//     PlcTask Inputs/m01_rs3_r1._05_TT_01_Error <-> TC Channel 1/Status/Error
//     PlcTask Inputs/m01_rs3_r1._05_TT_03_Error <-> TC Channel 2/Status/Error
//     PlcTask Inputs/m01_rs3_r1._06_TT_01_Error <-> TC Channel 3/Status/Error
//     PlcTask Inputs/m01_rs3_r1._06_TT_03_Error <-> TC Channel 4/Status/Error
//     PlcTask Inputs/m01_rs3_r1._07_TT_01_Error <-> TC Channel 5/Status/Error
//     PlcTask Inputs/m01_rs3_r1._07_TT_03_Error <-> TC Channel 6/Status/Error
//     PlcTask Inputs/m01_rs3_r1._08_TT_01_Error <-> TC Channel 7/Status/Error
//     PlcTask Inputs/m01_rs3_r1._08_TT_03_Error <-> TC Channel 8/Status/Error
//   Phase0/Phase0 Instance <-> Device 4 (EtherCAT)/Term 1 Server Rack (EK1100)/Term 3 To DAC Mod and BOP PWR (EK1122)/Term 4 Main DAC Panel(EK1100)/Term 116 To RS3 (EK1122)/Term 117  RS3 INST Top Row (EK1100)/Term 144 (EL3318)
//     PlcTask Inputs/m01_rs3_r1._09_TT_01 <-> TC Channel 1/Value
//     PlcTask Inputs/m01_rs3_r1._09_TT_03 <-> TC Channel 2/Value
//     PlcTask Inputs/m01_rs3_r1._10_TT_01 <-> TC Channel 3/Value
//     PlcTask Inputs/m01_rs3_r1._10_TT_03 <-> TC Channel 4/Value
//     PlcTask Inputs/m01_rs3_r1._11_TT_01 <-> TC Channel 5/Value
//     PlcTask Inputs/m01_rs3_r1._11_TT_03 <-> TC Channel 6/Value
//     PlcTask Inputs/m01_rs3_r1._12_TT_01 <-> TC Channel 7/Value
//     PlcTask Inputs/m01_rs3_r1._12_TT_03 <-> TC Channel 8/Value
//     PlcTask Inputs/m01_rs3_r1._09_TT_01_Error <-> TC Channel 1/Status/Error
//     PlcTask Inputs/m01_rs3_r1._09_TT_03_Error <-> TC Channel 2/Status/Error
//     PlcTask Inputs/m01_rs3_r1._10_TT_01_Error <-> TC Channel 3/Status/Error
//     PlcTask Inputs/m01_rs3_r1._10_TT_03_Error <-> TC Channel 4/Status/Error
//     PlcTask Inputs/m01_rs3_r1._11_TT_01_Error <-> TC Channel 5/Status/Error
//     PlcTask Inputs/m01_rs3_r1._11_TT_03_Error <-> TC Channel 6/Status/Error
//     PlcTask Inputs/m01_rs3_r1._12_TT_01_Error <-> TC Channel 7/Status/Error
//     PlcTask Inputs/m01_rs3_r1._12_TT_03_Error <-> TC Channel 8/Status/Error
//   Phase0/Phase0 Instance <-> Device 4 (EtherCAT)/Term 1 Server Rack (EK1100)/Term 3 To DAC Mod and BOP PWR (EK1122)/Term 4 Main DAC Panel(EK1100)/Term 116 To RS3 (EK1122)/Term 117  RS3 INST Top Row (EK1100)/Term 145 (EL3318)
//     PlcTask Inputs/m01_rs3_r3._01_TT_01 <-> TC Channel 1/Value
//     PlcTask Inputs/m01_rs3_r3._01_TT_03 <-> TC Channel 2/Value
//     PlcTask Inputs/m01_rs3_r3._02_TT_01 <-> TC Channel 3/Value
//     PlcTask Inputs/m01_rs3_r3._02_TT_03 <-> TC Channel 4/Value
//     PlcTask Inputs/m01_rs3_r3._03_TT_01 <-> TC Channel 5/Value
//     PlcTask Inputs/m01_rs3_r3._03_TT_03 <-> TC Channel 6/Value
//     PlcTask Inputs/m01_rs3_r3._04_TT_01 <-> TC Channel 7/Value
//     PlcTask Inputs/m01_rs3_r3._04_TT_03 <-> TC Channel 8/Value
//     PlcTask Inputs/m01_rs3_r3._01_TT_01_Error <-> TC Channel 1/Status/Error
//     PlcTask Inputs/m01_rs3_r3._01_TT_03_Error <-> TC Channel 2/Status/Error
//     PlcTask Inputs/m01_rs3_r3._02_TT_01_Error <-> TC Channel 3/Status/Error
//     PlcTask Inputs/m01_rs3_r3._02_TT_03_Error <-> TC Channel 4/Status/Error
//     PlcTask Inputs/m01_rs3_r3._03_TT_01_Error <-> TC Channel 5/Status/Error
//     PlcTask Inputs/m01_rs3_r3._03_TT_03_Error <-> TC Channel 6/Status/Error
//     PlcTask Inputs/m01_rs3_r3._04_TT_01_Error <-> TC Channel 7/Status/Error
//     PlcTask Inputs/m01_rs3_r3._04_TT_03_Error <-> TC Channel 8/Status/Error
//   Phase0/Phase0 Instance <-> Device 4 (EtherCAT)/Term 1 Server Rack (EK1100)/Term 3 To DAC Mod and BOP PWR (EK1122)/Term 4 Main DAC Panel(EK1100)/Term 116 To RS3 (EK1122)/Term 117  RS3 INST Top Row (EK1100)/Term 146 (EL3318)
//     PlcTask Inputs/m01_rs3_r3._05_TT_01 <-> TC Channel 1/Value
//     PlcTask Inputs/m01_rs3_r3._05_TT_03 <-> TC Channel 2/Value
//     PlcTask Inputs/m01_rs3_r3._06_TT_01 <-> TC Channel 3/Value
//     PlcTask Inputs/m01_rs3_r3._06_TT_03 <-> TC Channel 4/Value
//     PlcTask Inputs/m01_rs3_r3._07_TT_01 <-> TC Channel 5/Value
//     PlcTask Inputs/m01_rs3_r3._07_TT_03 <-> TC Channel 6/Value
//     PlcTask Inputs/m01_rs3_r3._08_TT_01 <-> TC Channel 7/Value
//     PlcTask Inputs/m01_rs3_r3._08_TT_03 <-> TC Channel 8/Value
//     PlcTask Inputs/m01_rs3_r3._05_TT_01_Error <-> TC Channel 1/Status/Error
//     PlcTask Inputs/m01_rs3_r3._05_TT_03_Error <-> TC Channel 2/Status/Error
//     PlcTask Inputs/m01_rs3_r3._06_TT_01_Error <-> TC Channel 3/Status/Error
//     PlcTask Inputs/m01_rs3_r3._06_TT_03_Error <-> TC Channel 4/Status/Error
//     PlcTask Inputs/m01_rs3_r3._07_TT_01_Error <-> TC Channel 5/Status/Error
//     PlcTask Inputs/m01_rs3_r3._07_TT_03_Error <-> TC Channel 6/Status/Error
//     PlcTask Inputs/m01_rs3_r3._08_TT_01_Error <-> TC Channel 7/Status/Error
//     PlcTask Inputs/m01_rs3_r3._08_TT_03_Error <-> TC Channel 8/Status/Error
//   Phase0/Phase0 Instance <-> Device 4 (EtherCAT)/Term 1 Server Rack (EK1100)/Term 3 To DAC Mod and BOP PWR (EK1122)/Term 4 Main DAC Panel(EK1100)/Term 116 To RS3 (EK1122)/Term 117  RS3 INST Top Row (EK1100)/Term 147 (EL3318)
//     PlcTask Inputs/m01_rs3_r3._09_TT_01 <-> TC Channel 1/Value
//     PlcTask Inputs/m01_rs3_r3._09_TT_03 <-> TC Channel 2/Value
//     PlcTask Inputs/m01_rs3_r3._10_TT_01 <-> TC Channel 3/Value
//     PlcTask Inputs/m01_rs3_r3._10_TT_03 <-> TC Channel 4/Value
//     PlcTask Inputs/m01_rs3_r3._11_TT_01 <-> TC Channel 5/Value
//     PlcTask Inputs/m01_rs3_r3._11_TT_03 <-> TC Channel 6/Value
//     PlcTask Inputs/m01_rs3_r3._12_TT_01 <-> TC Channel 7/Value
//     PlcTask Inputs/m01_rs3_r3._12_TT_03 <-> TC Channel 8/Value
//     PlcTask Inputs/m01_rs3_r3._09_TT_01_Error <-> TC Channel 1/Status/Error
//     PlcTask Inputs/m01_rs3_r3._09_TT_03_Error <-> TC Channel 2/Status/Error
//     PlcTask Inputs/m01_rs3_r3._10_TT_01_Error <-> TC Channel 3/Status/Error
//     PlcTask Inputs/m01_rs3_r3._10_TT_03_Error <-> TC Channel 4/Status/Error
//     PlcTask Inputs/m01_rs3_r3._11_TT_01_Error <-> TC Channel 5/Status/Error
//     PlcTask Inputs/m01_rs3_r3._11_TT_03_Error <-> TC Channel 6/Status/Error
//     PlcTask Inputs/m01_rs3_r3._12_TT_01_Error <-> TC Channel 7/Status/Error
//     PlcTask Inputs/m01_rs3_r3._12_TT_03_Error <-> TC Channel 8/Status/Error
//   Phase0/Phase0 Instance <-> Device 4 (EtherCAT)/Term 1 Server Rack (EK1100)/Term 3 To DAC Mod and BOP PWR (EK1122)/Term 4 Main DAC Panel(EK1100)/Term 116 To RS3 (EK1122)/Term 117  RS3 INST Top Row (EK1100)/Term 149 (EL3318)
//     PlcTask Inputs/m01_rs3_r2._01_TT_01 <-> TC Channel 1/Value
//     PlcTask Inputs/m01_rs3_r2._01_TT_03 <-> TC Channel 2/Value
//     PlcTask Inputs/m01_rs3_r2._02_TT_01 <-> TC Channel 3/Value
//     PlcTask Inputs/m01_rs3_r2._02_TT_03 <-> TC Channel 4/Value
//     PlcTask Inputs/m01_rs3_r2._03_TT_01 <-> TC Channel 5/Value
//     PlcTask Inputs/m01_rs3_r2._03_TT_03 <-> TC Channel 6/Value
//     PlcTask Inputs/m01_rs3_r2._04_TT_01 <-> TC Channel 7/Value
//     PlcTask Inputs/m01_rs3_r2._04_TT_03 <-> TC Channel 8/Value
//     PlcTask Inputs/m01_rs3_r2._01_TT_01_Error <-> TC Channel 1/Status/Error
//     PlcTask Inputs/m01_rs3_r2._01_TT_03_Error <-> TC Channel 2/Status/Error
//     PlcTask Inputs/m01_rs3_r2._02_TT_01_Error <-> TC Channel 3/Status/Error
//     PlcTask Inputs/m01_rs3_r2._02_TT_03_Error <-> TC Channel 4/Status/Error
//     PlcTask Inputs/m01_rs3_r2._03_TT_01_Error <-> TC Channel 5/Status/Error
//     PlcTask Inputs/m01_rs3_r2._03_TT_03_Error <-> TC Channel 6/Status/Error
//     PlcTask Inputs/m01_rs3_r2._04_TT_01_Error <-> TC Channel 7/Status/Error
//     PlcTask Inputs/m01_rs3_r2._04_TT_03_Error <-> TC Channel 8/Status/Error
//   Phase0/Phase0 Instance <-> Device 4 (EtherCAT)/Term 1 Server Rack (EK1100)/Term 3 To DAC Mod and BOP PWR (EK1122)/Term 4 Main DAC Panel(EK1100)/Term 116 To RS3 (EK1122)/Term 117  RS3 INST Top Row (EK1100)/Term 150 (EL3318)
//     PlcTask Inputs/m01_rs3_r2._05_TT_01 <-> TC Channel 1/Value
//     PlcTask Inputs/m01_rs3_r2._05_TT_03 <-> TC Channel 2/Value
//     PlcTask Inputs/m01_rs3_r2._06_TT_01 <-> TC Channel 3/Value
//     PlcTask Inputs/m01_rs3_r2._06_TT_03 <-> TC Channel 4/Value
//     PlcTask Inputs/m01_rs3_r2._07_TT_01 <-> TC Channel 5/Value
//     PlcTask Inputs/m01_rs3_r2._07_TT_03 <-> TC Channel 6/Value
//     PlcTask Inputs/m01_rs3_r2._08_TT_01 <-> TC Channel 7/Value
//     PlcTask Inputs/m01_rs3_r2._08_TT_03 <-> TC Channel 8/Value
//     PlcTask Inputs/m01_rs3_r2._05_TT_01_Error <-> TC Channel 1/Status/Error
//     PlcTask Inputs/m01_rs3_r2._05_TT_03_Error <-> TC Channel 2/Status/Error
//     PlcTask Inputs/m01_rs3_r2._06_TT_01_Error <-> TC Channel 3/Status/Error
//     PlcTask Inputs/m01_rs3_r2._06_TT_03_Error <-> TC Channel 4/Status/Error
//     PlcTask Inputs/m01_rs3_r2._07_TT_01_Error <-> TC Channel 5/Status/Error
//     PlcTask Inputs/m01_rs3_r2._07_TT_03_Error <-> TC Channel 6/Status/Error
//     PlcTask Inputs/m01_rs3_r2._08_TT_01_Error <-> TC Channel 7/Status/Error
//     PlcTask Inputs/m01_rs3_r2._08_TT_03_Error <-> TC Channel 8/Status/Error
//   Phase0/Phase0 Instance <-> Device 4 (EtherCAT)/Term 1 Server Rack (EK1100)/Term 3 To DAC Mod and BOP PWR (EK1122)/Term 4 Main DAC Panel(EK1100)/Term 116 To RS3 (EK1122)/Term 117  RS3 INST Top Row (EK1100)/Term 151 (EL3318)
//     PlcTask Inputs/m01_rs3_r2._09_TT_01 <-> TC Channel 1/Value
//     PlcTask Inputs/m01_rs3_r2._09_TT_03 <-> TC Channel 2/Value
//     PlcTask Inputs/m01_rs3_r2._10_TT_01 <-> TC Channel 3/Value
//     PlcTask Inputs/m01_rs3_r2._10_TT_03 <-> TC Channel 4/Value
//     PlcTask Inputs/m01_rs3_r2._11_TT_01 <-> TC Channel 5/Value
//     PlcTask Inputs/m01_rs3_r2._11_TT_03 <-> TC Channel 6/Value
//     PlcTask Inputs/m01_rs3_r2._12_TT_01 <-> TC Channel 7/Value
//     PlcTask Inputs/m01_rs3_r2._12_TT_03 <-> TC Channel 8/Value
//     PlcTask Inputs/m01_rs3_r2._09_TT_01_Error <-> TC Channel 1/Status/Error
//     PlcTask Inputs/m01_rs3_r2._09_TT_03_Error <-> TC Channel 2/Status/Error
//     PlcTask Inputs/m01_rs3_r2._10_TT_01_Error <-> TC Channel 3/Status/Error
//     PlcTask Inputs/m01_rs3_r2._10_TT_03_Error <-> TC Channel 4/Status/Error
//     PlcTask Inputs/m01_rs3_r2._11_TT_01_Error <-> TC Channel 5/Status/Error
//     PlcTask Inputs/m01_rs3_r2._11_TT_03_Error <-> TC Channel 6/Status/Error
//     PlcTask Inputs/m01_rs3_r2._12_TT_01_Error <-> TC Channel 7/Status/Error
//     PlcTask Inputs/m01_rs3_r2._12_TT_03_Error <-> TC Channel 8/Status/Error
//   Phase0/Phase0 Instance <-> Device 4 (EtherCAT)/Term 1 Server Rack (EK1100)/Term 3 To DAC Mod and BOP PWR (EK1122)/Term 4 Main DAC Panel(EK1100)/Term 116 To RS3 (EK1122)/Term 117  RS3 INST Top Row (EK1100)/Term 152 (EL3318)
//     PlcTask Inputs/m01_rs3_r4._01_TT_01 <-> TC Channel 1/Value
//     PlcTask Inputs/m01_rs3_r4._01_TT_03 <-> TC Channel 2/Value
//     PlcTask Inputs/m01_rs3_r4._02_TT_01 <-> TC Channel 3/Value
//     PlcTask Inputs/m01_rs3_r4._02_TT_03 <-> TC Channel 4/Value
//     PlcTask Inputs/m01_rs3_r4._03_TT_01 <-> TC Channel 5/Value
//     PlcTask Inputs/m01_rs3_r4._03_TT_03 <-> TC Channel 6/Value
//     PlcTask Inputs/m01_rs3_r4._04_TT_01 <-> TC Channel 7/Value
//     PlcTask Inputs/m01_rs3_r4._04_TT_03 <-> TC Channel 8/Value
//     PlcTask Inputs/m01_rs3_r4._01_TT_01_Error <-> TC Channel 1/Status/Error
//     PlcTask Inputs/m01_rs3_r4._01_TT_03_Error <-> TC Channel 2/Status/Error
//     PlcTask Inputs/m01_rs3_r4._02_TT_01_Error <-> TC Channel 3/Status/Error
//     PlcTask Inputs/m01_rs3_r4._02_TT_03_Error <-> TC Channel 4/Status/Error
//     PlcTask Inputs/m01_rs3_r4._03_TT_01_Error <-> TC Channel 5/Status/Error
//     PlcTask Inputs/m01_rs3_r4._03_TT_03_Error <-> TC Channel 6/Status/Error
//     PlcTask Inputs/m01_rs3_r4._04_TT_01_Error <-> TC Channel 7/Status/Error
//     PlcTask Inputs/m01_rs3_r4._04_TT_03_Error <-> TC Channel 8/Status/Error
//   Phase0/Phase0 Instance <-> Device 4 (EtherCAT)/Term 1 Server Rack (EK1100)/Term 3 To DAC Mod and BOP PWR (EK1122)/Term 4 Main DAC Panel(EK1100)/Term 116 To RS3 (EK1122)/Term 117  RS3 INST Top Row (EK1100)/Term 153 (EL3318)
//     PlcTask Inputs/m01_rs3_r4._05_TT_01 <-> TC Channel 1/Value
//     PlcTask Inputs/m01_rs3_r4._05_TT_03 <-> TC Channel 2/Value
//     PlcTask Inputs/m01_rs3_r4._06_TT_01 <-> TC Channel 3/Value
//     PlcTask Inputs/m01_rs3_r4._06_TT_03 <-> TC Channel 4/Value
//     PlcTask Inputs/m01_rs3_r4._07_TT_01 <-> TC Channel 5/Value
//     PlcTask Inputs/m01_rs3_r4._07_TT_03 <-> TC Channel 6/Value
//     PlcTask Inputs/m01_rs3_r4._08_TT_01 <-> TC Channel 7/Value
//     PlcTask Inputs/m01_rs3_r4._08_TT_03 <-> TC Channel 8/Value
//     PlcTask Inputs/m01_rs3_r4._05_TT_01_Error <-> TC Channel 1/Status/Error
//     PlcTask Inputs/m01_rs3_r4._05_TT_03_Error <-> TC Channel 2/Status/Error
//     PlcTask Inputs/m01_rs3_r4._06_TT_01_Error <-> TC Channel 3/Status/Error
//     PlcTask Inputs/m01_rs3_r4._06_TT_03_Error <-> TC Channel 4/Status/Error
//     PlcTask Inputs/m01_rs3_r4._07_TT_01_Error <-> TC Channel 5/Status/Error
//     PlcTask Inputs/m01_rs3_r4._07_TT_03_Error <-> TC Channel 6/Status/Error
//     PlcTask Inputs/m01_rs3_r4._08_TT_01_Error <-> TC Channel 7/Status/Error
//     PlcTask Inputs/m01_rs3_r4._08_TT_03_Error <-> TC Channel 8/Status/Error
//   Phase0/Phase0 Instance <-> Device 4 (EtherCAT)/Term 1 Server Rack (EK1100)/Term 3 To DAC Mod and BOP PWR (EK1122)/Term 4 Main DAC Panel(EK1100)/Term 116 To RS3 (EK1122)/Term 117  RS3 INST Top Row (EK1100)/Term 154 (EL3318)
//     PlcTask Inputs/m01_rs3_r4._09_TT_01 <-> TC Channel 1/Value
//     PlcTask Inputs/m01_rs3_r4._09_TT_03 <-> TC Channel 2/Value
//     PlcTask Inputs/m01_rs3_r4._10_TT_01 <-> TC Channel 3/Value
//     PlcTask Inputs/m01_rs3_r4._10_TT_03 <-> TC Channel 4/Value
//     PlcTask Inputs/m01_rs3_r4._11_TT_01 <-> TC Channel 5/Value
//     PlcTask Inputs/m01_rs3_r4._11_TT_03 <-> TC Channel 6/Value
//     PlcTask Inputs/m01_rs3_r4._12_TT_01 <-> TC Channel 7/Value
//     PlcTask Inputs/m01_rs3_r4._12_TT_03 <-> TC Channel 8/Value
//     PlcTask Inputs/m01_rs3_r4._09_TT_01_Error <-> TC Channel 1/Status/Error
//     PlcTask Inputs/m01_rs3_r4._09_TT_03_Error <-> TC Channel 2/Status/Error
//     PlcTask Inputs/m01_rs3_r4._10_TT_01_Error <-> TC Channel 3/Status/Error
//     PlcTask Inputs/m01_rs3_r4._10_TT_03_Error <-> TC Channel 4/Status/Error
//     PlcTask Inputs/m01_rs3_r4._11_TT_01_Error <-> TC Channel 5/Status/Error
//     PlcTask Inputs/m01_rs3_r4._11_TT_03_Error <-> TC Channel 6/Status/Error
//     PlcTask Inputs/m01_rs3_r4._12_TT_01_Error <-> TC Channel 7/Status/Error
//     PlcTask Inputs/m01_rs3_r4._12_TT_03_Error <-> TC Channel 8/Status/Error
//   Phase0/Phase0 Instance <-> Device 4 (EtherCAT)/Term 1 Server Rack (EK1100)/Term 3 To DAC Mod and BOP PWR (EK1122)/Term 4 Main DAC Panel(EK1100)/Term 116 To RS3 (EK1122)/Term 117  RS3 INST Top Row (EK1100)/Term 156 (EL3214)
//     PlcTask Inputs/m01_rs3_r1.TT_05 <-> RTD Inputs Channel 1/Value
//     PlcTask Inputs/m01_rs3_r2.TT_05 <-> RTD Inputs Channel 3/Value
//     PlcTask Inputs/m01_rs3_r3.TT_05 <-> RTD Inputs Channel 2/Value
//     PlcTask Inputs/m01_rs3_r4.TT_05 <-> RTD Inputs Channel 4/Value
//     PlcTask Inputs/m01_rs3_r1.reactor_wall_temp_error <-> RTD Inputs Channel 1/Status/Error
//     PlcTask Inputs/m01_rs3_r2.reactor_wall_temp_error <-> RTD Inputs Channel 3/Status/Error
//     PlcTask Inputs/m01_rs3_r3.reactor_wall_temp_error <-> RTD Inputs Channel 2/Status/Error
//     PlcTask Inputs/m01_rs3_r4.reactor_wall_temp_error <-> RTD Inputs Channel 4/Status/Error
//   Phase0/Phase0 Instance <-> Device 4 (EtherCAT)/Term 1 Server Rack (EK1100)/Term 3 To DAC Mod and BOP PWR (EK1122)/Term 4 Main DAC Panel(EK1100)/Term 116 To RS3 (EK1122)/Term 117  RS3 INST Top Row (EK1100)/Term 157 (EL3214)
//     PlcTask Inputs/m01_rs3_r1.TT_06 <-> RTD Inputs Channel 1/Value
//     PlcTask Inputs/m01_rs3_r2.TT_06 <-> RTD Inputs Channel 3/Value
//     PlcTask Inputs/m01_rs3_r3.TT_06 <-> RTD Inputs Channel 2/Value
//     PlcTask Inputs/m01_rs3_r4.TT_06 <-> RTD Inputs Channel 4/Value
//     PlcTask Inputs/m01_rs3_r1.outlet_line_temp_error <-> RTD Inputs Channel 1/Status/Error
//     PlcTask Inputs/m01_rs3_r2.outlet_line_temp_error <-> RTD Inputs Channel 3/Status/Error
//     PlcTask Inputs/m01_rs3_r3.outlet_line_temp_error <-> RTD Inputs Channel 2/Status/Error
//     PlcTask Inputs/m01_rs3_r4.outlet_line_temp_error <-> RTD Inputs Channel 4/Status/Error
//   Phase0/Phase0 Instance <-> Device 4 (EtherCAT)/Term 1 Server Rack (EK1100)/Term 3 To DAC Mod and BOP PWR (EK1122)/Term 4 Main DAC Panel(EK1100)/Term 116 To RS3 (EK1122)/Term 159  RS3 INST Bot Row (EK1100)/Term 160 (EL2008)
//     PlcTask Outputs/m01_rs3_r1.XV_01_Door_Close_Solenoid_Valve <-> Channel 2/Output
//     PlcTask Outputs/m01_rs3_r1.XV_03_Door_Close_Solenoid_Valve <-> Channel 4/Output
//     PlcTask Outputs/m01_rs3_r3.XV_01_Door_Close_Solenoid_Valve <-> Channel 6/Output
//     PlcTask Outputs/m01_rs3_r3.XV_03_Door_Close_Solenoid_Valve <-> Channel 8/Output
//     PlcTask Outputs/m01_rs3_r1.XV_01_Door_Open_Solenoid_Valve <-> Channel 1/Output
//     PlcTask Outputs/m01_rs3_r1.XV_03_Door_Open_Solenoid_Valve <-> Channel 3/Output
//     PlcTask Outputs/m01_rs3_r3.XV_01_Door_Open_Solenoid_Valve <-> Channel 5/Output
//     PlcTask Outputs/m01_rs3_r3.XV_03_Door_Open_Solenoid_Valve <-> Channel 7/Output
//   Phase0/Phase0 Instance <-> Device 4 (EtherCAT)/Term 1 Server Rack (EK1100)/Term 3 To DAC Mod and BOP PWR (EK1122)/Term 4 Main DAC Panel(EK1100)/Term 116 To RS3 (EK1122)/Term 159  RS3 INST Bot Row (EK1100)/Term 161 (EL2008)
//     PlcTask Outputs/m01_rs3_r2.XV_01_Door_Close_Solenoid_Valve <-> Channel 2/Output
//     PlcTask Outputs/m01_rs3_r2.XV_03_Door_Close_Solenoid_Valve <-> Channel 4/Output
//     PlcTask Outputs/m01_rs3_r4.XV_01_Door_Close_Solenoid_Valve <-> Channel 6/Output
//     PlcTask Outputs/m01_rs3_r4.XV_03_Door_Close_Solenoid_Valve <-> Channel 8/Output
//     PlcTask Outputs/m01_rs3_r2.XV_01_Door_Open_Solenoid_Valve <-> Channel 1/Output
//     PlcTask Outputs/m01_rs3_r2.XV_03_Door_Open_Solenoid_Valve <-> Channel 3/Output
//     PlcTask Outputs/m01_rs3_r4.XV_01_Door_Open_Solenoid_Valve <-> Channel 5/Output
//     PlcTask Outputs/m01_rs3_r4.XV_03_Door_Open_Solenoid_Valve <-> Channel 7/Output
//   Phase0/Phase0 Instance <-> Device 4 (EtherCAT)/Term 1 Server Rack (EK1100)/Term 3 To DAC Mod and BOP PWR (EK1122)/Term 4 Main DAC Panel(EK1100)/Term 116 To RS3 (EK1122)/Term 159  RS3 INST Bot Row (EK1100)/Term 163  To RS3 VFDs (EK1122)/Box 164 RS3 VFD1 (Commander C300 Open Loop)
//     PlcTask Inputs/m01_rs3_r1.fan_vfd_current <-> Transmit PDO Mapping 6/vfd output current param 04_001
//     PlcTask Inputs/m01_rs3_r1.fan_vfd_ecat_state <-> WcState/WcState
//     PlcTask Inputs/m01_rs3_r1.fan_vfd_status <-> Transmit PDO Mapping 6/Status word
//     PlcTask Inputs/m01_rs3_r1.fan_vfd_temp <-> Transmit PDO Mapping 6/inverter temp 07_034
//     PlcTask Inputs/m01_rs3_r1.fan_vfd_velocity <-> Transmit PDO Mapping 6/vl velocity actual value
//     PlcTask Outputs/m01_rs3_r1.fan_vfd_control <-> Receive PDO Mapping 6/Control word
//     PlcTask Outputs/m01_rs3_r1.fan_vfd_target_vel <-> Receive PDO Mapping 6/vl target velocity
//   Phase0/Phase0 Instance <-> Device 4 (EtherCAT)/Term 1 Server Rack (EK1100)/Term 3 To DAC Mod and BOP PWR (EK1122)/Term 4 Main DAC Panel(EK1100)/Term 116 To RS3 (EK1122)/Term 159  RS3 INST Bot Row (EK1100)/Term 163  To RS3 VFDs (EK1122)/Box 165 RS3 VFD2 (Commander C300 Open Loop)
//     PlcTask Inputs/m01_rs3_r2.fan_vfd_current <-> Transmit PDO Mapping 6/vfd output current param 04_001
//     PlcTask Inputs/m01_rs3_r2.fan_vfd_ecat_state <-> WcState/WcState
//     PlcTask Inputs/m01_rs3_r2.fan_vfd_status <-> Transmit PDO Mapping 6/Status word
//     PlcTask Inputs/m01_rs3_r2.fan_vfd_velocity <-> Transmit PDO Mapping 6/vl velocity actual value
//     PlcTask Outputs/m01_rs3_r2.fan_vfd_control <-> Receive PDO Mapping 6/Control word
//     PlcTask Outputs/m01_rs3_r2.fan_vfd_target_vel <-> Receive PDO Mapping 6/vl target velocity
//   Phase0/Phase0 Instance <-> Device 4 (EtherCAT)/Term 1 Server Rack (EK1100)/Term 3 To DAC Mod and BOP PWR (EK1122)/Term 4 Main DAC Panel(EK1100)/Term 116 To RS3 (EK1122)/Term 159  RS3 INST Bot Row (EK1100)/Term 163  To RS3 VFDs (EK1122)/Box 166 RS3 VFD3 (Commander C300 Open Loop)
//     PlcTask Inputs/m01_rs3_r3.fan_vfd_current <-> Transmit PDO Mapping 6/vfd output current param 04_001
//     PlcTask Inputs/m01_rs3_r3.fan_vfd_ecat_state <-> WcState/WcState
//     PlcTask Inputs/m01_rs3_r3.fan_vfd_status <-> Transmit PDO Mapping 6/Status word
//     PlcTask Inputs/m01_rs3_r3.fan_vfd_velocity <-> Transmit PDO Mapping 6/vl velocity actual value
//     PlcTask Outputs/m01_rs3_r3.fan_vfd_control <-> Receive PDO Mapping 6/Control word
//     PlcTask Outputs/m01_rs3_r3.fan_vfd_target_vel <-> Receive PDO Mapping 6/vl target velocity
//   Phase0/Phase0 Instance <-> Device 4 (EtherCAT)/Term 1 Server Rack (EK1100)/Term 3 To DAC Mod and BOP PWR (EK1122)/Term 4 Main DAC Panel(EK1100)/Term 116 To RS3 (EK1122)/Term 159  RS3 INST Bot Row (EK1100)/Term 163  To RS3 VFDs (EK1122)/Box 167 RS3 VFD4 (Commander C300 Open Loop)
//     PlcTask Inputs/m01_rs3_r4.fan_vfd_current <-> Transmit PDO Mapping 6/vfd output current param 04_001
//     PlcTask Inputs/m01_rs3_r4.fan_vfd_ecat_state <-> WcState/WcState
//     PlcTask Inputs/m01_rs3_r4.fan_vfd_status <-> Transmit PDO Mapping 6/Status word
//     PlcTask Inputs/m01_rs3_r4.fan_vfd_velocity <-> Transmit PDO Mapping 6/vl velocity actual value
//     PlcTask Outputs/m01_rs3_r4.fan_vfd_control <-> Receive PDO Mapping 6/Control word
//     PlcTask Outputs/m01_rs3_r4.fan_vfd_target_vel <-> Receive PDO Mapping 6/vl target velocity
//   Phase0/Phase0 Instance <-> Device 4 (EtherCAT)/Term 1 Server Rack (EK1100)/Term 3 To DAC Mod and BOP PWR (EK1122)/Term 4 Main DAC Panel(EK1100)/Term 5 (EL1008)
//     PlcTask Inputs/m01.condensate_from_cooling_and_purge_lines_lsh <-> Channel 2/Input
//     PlcTask Inputs/m01.condensate_from_cooling_and_purge_lines_lsl <-> Channel 1/Input
//   Phase0/Phase0 Instance <-> Device 4 (EtherCAT)/Term 1 Server Rack (EK1100)/Term 3 To DAC Mod and BOP PWR (EK1122)/Term 4 Main DAC Panel(EK1100)/Term 6 (EL1008)
//     PlcTask Inputs/m01_rs1.circuit_breaker_nc_feedback <-> Channel 4/Input
//     PlcTask Inputs/m01_rs2.circuit_breaker_nc_feedback <-> Channel 6/Input
//     PlcTask Inputs/m01_rs3.circuit_breaker_nc_feedback <-> Channel 2/Input
//     PlcTask Inputs/m01_rs1.circuit_breaker_no_feedback <-> Channel 3/Input
//     PlcTask Inputs/m01_rs2.circuit_breaker_no_feedback <-> Channel 5/Input
//     PlcTask Inputs/m01_rs3.circuit_breaker_no_feedback <-> Channel 1/Input
//   Phase0/Phase0 Instance <-> Device 4 (EtherCAT)/Term 1 Server Rack (EK1100)/Term 3 To DAC Mod and BOP PWR (EK1122)/Term 4 Main DAC Panel(EK1100)/Term 63 To RS2 (EK1122)/Term 106  RS2 INST Bot Row (EK1100)/Term 107 (EL2008)
//     PlcTask Outputs/m01_rs2_r1.XV_01_Door_Close_Solenoid_Valve <-> Channel 2/Output
//     PlcTask Outputs/m01_rs2_r1.XV_03_Door_Close_Solenoid_Valve <-> Channel 4/Output
//     PlcTask Outputs/m01_rs2_r3.XV_01_Door_Close_Solenoid_Valve <-> Channel 6/Output
//     PlcTask Outputs/m01_rs2_r3.XV_03_Door_Close_Solenoid_Valve <-> Channel 8/Output
//     PlcTask Outputs/m01_rs2_r1.XV_01_Door_Open_Solenoid_Valve <-> Channel 1/Output
//     PlcTask Outputs/m01_rs2_r1.XV_03_Door_Open_Solenoid_Valve <-> Channel 3/Output
//     PlcTask Outputs/m01_rs2_r3.XV_01_Door_Open_Solenoid_Valve <-> Channel 5/Output
//     PlcTask Outputs/m01_rs2_r3.XV_03_Door_Open_Solenoid_Valve <-> Channel 7/Output
//   Phase0/Phase0 Instance <-> Device 4 (EtherCAT)/Term 1 Server Rack (EK1100)/Term 3 To DAC Mod and BOP PWR (EK1122)/Term 4 Main DAC Panel(EK1100)/Term 63 To RS2 (EK1122)/Term 106  RS2 INST Bot Row (EK1100)/Term 108 (EL2008)
//     PlcTask Outputs/m01_rs2_r2.XV_01_Door_Close_Solenoid_Valve <-> Channel 2/Output
//     PlcTask Outputs/m01_rs2_r2.XV_03_Door_Close_Solenoid_Valve <-> Channel 4/Output
//     PlcTask Outputs/m01_rs2_r4.XV_01_Door_Close_Solenoid_Valve <-> Channel 6/Output
//     PlcTask Outputs/m01_rs2_r4.XV_03_Door_Close_Solenoid_Valve <-> Channel 8/Output
//     PlcTask Outputs/m01_rs2_r2.XV_01_Door_Open_Solenoid_Valve <-> Channel 1/Output
//     PlcTask Outputs/m01_rs2_r2.XV_03_Door_Open_Solenoid_Valve <-> Channel 3/Output
//     PlcTask Outputs/m01_rs2_r4.XV_01_Door_Open_Solenoid_Valve <-> Channel 5/Output
//     PlcTask Outputs/m01_rs2_r4.XV_03_Door_Open_Solenoid_Valve <-> Channel 7/Output
//   Phase0/Phase0 Instance <-> Device 4 (EtherCAT)/Term 1 Server Rack (EK1100)/Term 3 To DAC Mod and BOP PWR (EK1122)/Term 4 Main DAC Panel(EK1100)/Term 63 To RS2 (EK1122)/Term 106  RS2 INST Bot Row (EK1100)/Term 110  To RS2 VFDs (EK1122)/Box 111 RS2 VFD1 (Commander C300 Open Loop)
//     PlcTask Inputs/m01_rs2_r1.fan_vfd_current <-> Transmit PDO Mapping 6/vfd output current param 04_001
//     PlcTask Inputs/m01_rs2_r1.fan_vfd_ecat_state <-> WcState/WcState
//     PlcTask Inputs/m01_rs2_r1.fan_vfd_status <-> Transmit PDO Mapping 6/Status word
//     PlcTask Inputs/m01_rs2_r1.fan_vfd_temp <-> Transmit PDO Mapping 6/inverter temp 07_034
//     PlcTask Inputs/m01_rs2_r1.fan_vfd_velocity <-> Transmit PDO Mapping 6/vl velocity actual value
//     PlcTask Outputs/m01_rs2_r1.fan_vfd_control <-> Receive PDO Mapping 6/Control word
//     PlcTask Outputs/m01_rs2_r1.fan_vfd_target_vel <-> Receive PDO Mapping 6/vl target velocity
//   Phase0/Phase0 Instance <-> Device 4 (EtherCAT)/Term 1 Server Rack (EK1100)/Term 3 To DAC Mod and BOP PWR (EK1122)/Term 4 Main DAC Panel(EK1100)/Term 63 To RS2 (EK1122)/Term 106  RS2 INST Bot Row (EK1100)/Term 110  To RS2 VFDs (EK1122)/Box 112 RS2 VFD2 (Commander C300 Open Loop)
//     PlcTask Inputs/m01_rs2_r2.fan_vfd_current <-> Transmit PDO Mapping 6/vfd output current param 04_001
//     PlcTask Inputs/m01_rs2_r2.fan_vfd_ecat_state <-> WcState/WcState
//     PlcTask Inputs/m01_rs2_r2.fan_vfd_status <-> Transmit PDO Mapping 6/Status word
//     PlcTask Inputs/m01_rs2_r2.fan_vfd_velocity <-> Transmit PDO Mapping 6/vl velocity actual value
//     PlcTask Outputs/m01_rs2_r2.fan_vfd_control <-> Receive PDO Mapping 6/Control word
//     PlcTask Outputs/m01_rs2_r2.fan_vfd_target_vel <-> Receive PDO Mapping 6/vl target velocity
//   Phase0/Phase0 Instance <-> Device 4 (EtherCAT)/Term 1 Server Rack (EK1100)/Term 3 To DAC Mod and BOP PWR (EK1122)/Term 4 Main DAC Panel(EK1100)/Term 63 To RS2 (EK1122)/Term 106  RS2 INST Bot Row (EK1100)/Term 110  To RS2 VFDs (EK1122)/Box 113 RS2 VFD3 (Commander C300 Open Loop)
//     PlcTask Inputs/m01_rs2_r3.fan_vfd_current <-> Transmit PDO Mapping 6/vfd output current param 04_001
//     PlcTask Inputs/m01_rs2_r3.fan_vfd_ecat_state <-> WcState/WcState
//     PlcTask Inputs/m01_rs2_r3.fan_vfd_status <-> Transmit PDO Mapping 6/Status word
//     PlcTask Inputs/m01_rs2_r3.fan_vfd_velocity <-> Transmit PDO Mapping 6/vl velocity actual value
//     PlcTask Outputs/m01_rs2_r3.fan_vfd_control <-> Receive PDO Mapping 6/Control word
//     PlcTask Outputs/m01_rs2_r3.fan_vfd_target_vel <-> Receive PDO Mapping 6/vl target velocity
//   Phase0/Phase0 Instance <-> Device 4 (EtherCAT)/Term 1 Server Rack (EK1100)/Term 3 To DAC Mod and BOP PWR (EK1122)/Term 4 Main DAC Panel(EK1100)/Term 63 To RS2 (EK1122)/Term 106  RS2 INST Bot Row (EK1100)/Term 110  To RS2 VFDs (EK1122)/Box 114 RS2 VFD4 (Commander C300 Open Loop)
//     PlcTask Inputs/m01_rs2_r4.fan_vfd_current <-> Transmit PDO Mapping 6/vfd output current param 04_001
//     PlcTask Inputs/m01_rs2_r4.fan_vfd_ecat_state <-> WcState/WcState
//     PlcTask Inputs/m01_rs2_r4.fan_vfd_status <-> Transmit PDO Mapping 6/Status word
//     PlcTask Inputs/m01_rs2_r4.fan_vfd_velocity <-> Transmit PDO Mapping 6/vl velocity actual value
//     PlcTask Outputs/m01_rs2_r4.fan_vfd_control <-> Receive PDO Mapping 6/Control word
//     PlcTask Outputs/m01_rs2_r4.fan_vfd_target_vel <-> Receive PDO Mapping 6/vl target velocity
//   Phase0/Phase0 Instance <-> Device 4 (EtherCAT)/Term 1 Server Rack (EK1100)/Term 3 To DAC Mod and BOP PWR (EK1122)/Term 4 Main DAC Panel(EK1100)/Term 63 To RS2 (EK1122)/Term 64 RS2 INST Top Row (EK1100)/Term 100 (EL3318)
//     PlcTask Inputs/m01_rs2_r4._05_TT_01 <-> TC Channel 1/Value
//     PlcTask Inputs/m01_rs2_r4._05_TT_03 <-> TC Channel 2/Value
//     PlcTask Inputs/m01_rs2_r4._06_TT_01 <-> TC Channel 3/Value
//     PlcTask Inputs/m01_rs2_r4._06_TT_03 <-> TC Channel 4/Value
//     PlcTask Inputs/m01_rs2_r4._07_TT_01 <-> TC Channel 5/Value
//     PlcTask Inputs/m01_rs2_r4._07_TT_03 <-> TC Channel 6/Value
//     PlcTask Inputs/m01_rs2_r4._08_TT_01 <-> TC Channel 7/Value
//     PlcTask Inputs/m01_rs2_r4._08_TT_03 <-> TC Channel 8/Value
//     PlcTask Inputs/m01_rs2_r4._05_TT_01_Error <-> TC Channel 1/Status/Error
//     PlcTask Inputs/m01_rs2_r4._05_TT_03_Error <-> TC Channel 2/Status/Error
//     PlcTask Inputs/m01_rs2_r4._06_TT_01_Error <-> TC Channel 3/Status/Error
//     PlcTask Inputs/m01_rs2_r4._06_TT_03_Error <-> TC Channel 4/Status/Error
//     PlcTask Inputs/m01_rs2_r4._07_TT_01_Error <-> TC Channel 5/Status/Error
//     PlcTask Inputs/m01_rs2_r4._07_TT_03_Error <-> TC Channel 6/Status/Error
//     PlcTask Inputs/m01_rs2_r4._08_TT_01_Error <-> TC Channel 7/Status/Error
//     PlcTask Inputs/m01_rs2_r4._08_TT_03_Error <-> TC Channel 8/Status/Error
//   Phase0/Phase0 Instance <-> Device 4 (EtherCAT)/Term 1 Server Rack (EK1100)/Term 3 To DAC Mod and BOP PWR (EK1122)/Term 4 Main DAC Panel(EK1100)/Term 63 To RS2 (EK1122)/Term 64 RS2 INST Top Row (EK1100)/Term 101 (EL3318)
//     PlcTask Inputs/m01_rs2_r4._09_TT_01 <-> TC Channel 1/Value
//     PlcTask Inputs/m01_rs2_r4._09_TT_03 <-> TC Channel 2/Value
//     PlcTask Inputs/m01_rs2_r4._10_TT_01 <-> TC Channel 3/Value
//     PlcTask Inputs/m01_rs2_r4._10_TT_03 <-> TC Channel 4/Value
//     PlcTask Inputs/m01_rs2_r4._11_TT_01 <-> TC Channel 5/Value
//     PlcTask Inputs/m01_rs2_r4._11_TT_03 <-> TC Channel 6/Value
//     PlcTask Inputs/m01_rs2_r4._12_TT_01 <-> TC Channel 7/Value
//     PlcTask Inputs/m01_rs2_r4._12_TT_03 <-> TC Channel 8/Value
//     PlcTask Inputs/m01_rs2_r4._09_TT_01_Error <-> TC Channel 1/Status/Error
//     PlcTask Inputs/m01_rs2_r4._09_TT_03_Error <-> TC Channel 2/Status/Error
//     PlcTask Inputs/m01_rs2_r4._10_TT_01_Error <-> TC Channel 3/Status/Error
//     PlcTask Inputs/m01_rs2_r4._10_TT_03_Error <-> TC Channel 4/Status/Error
//     PlcTask Inputs/m01_rs2_r4._11_TT_01_Error <-> TC Channel 5/Status/Error
//     PlcTask Inputs/m01_rs2_r4._11_TT_03_Error <-> TC Channel 6/Status/Error
//     PlcTask Inputs/m01_rs2_r4._12_TT_01_Error <-> TC Channel 7/Status/Error
//     PlcTask Inputs/m01_rs2_r4._12_TT_03_Error <-> TC Channel 8/Status/Error
//   Phase0/Phase0 Instance <-> Device 4 (EtherCAT)/Term 1 Server Rack (EK1100)/Term 3 To DAC Mod and BOP PWR (EK1122)/Term 4 Main DAC Panel(EK1100)/Term 63 To RS2 (EK1122)/Term 64 RS2 INST Top Row (EK1100)/Term 103 (EL3214)
//     PlcTask Inputs/m01_rs2_r1.TT_05 <-> RTD Inputs Channel 1/Value
//     PlcTask Inputs/m01_rs2_r2.TT_05 <-> RTD Inputs Channel 3/Value
//     PlcTask Inputs/m01_rs2_r3.TT_05 <-> RTD Inputs Channel 2/Value
//     PlcTask Inputs/m01_rs2_r4.TT_05 <-> RTD Inputs Channel 4/Value
//     PlcTask Inputs/m01_rs2_r1.reactor_wall_temp_error <-> RTD Inputs Channel 1/Status/Error
//     PlcTask Inputs/m01_rs2_r2.reactor_wall_temp_error <-> RTD Inputs Channel 2/Status/Error
//     PlcTask Inputs/m01_rs2_r3.reactor_wall_temp_error <-> RTD Inputs Channel 3/Status/Error
//     PlcTask Inputs/m01_rs2_r4.reactor_wall_temp_error <-> RTD Inputs Channel 4/Status/Error
//   Phase0/Phase0 Instance <-> Device 4 (EtherCAT)/Term 1 Server Rack (EK1100)/Term 3 To DAC Mod and BOP PWR (EK1122)/Term 4 Main DAC Panel(EK1100)/Term 63 To RS2 (EK1122)/Term 64 RS2 INST Top Row (EK1100)/Term 104 (EL3214)
//     PlcTask Inputs/m01_rs2_r1.TT_06 <-> RTD Inputs Channel 1/Value
//     PlcTask Inputs/m01_rs2_r2.TT_06 <-> RTD Inputs Channel 3/Value
//     PlcTask Inputs/m01_rs2_r3.TT_06 <-> RTD Inputs Channel 2/Value
//     PlcTask Inputs/m01_rs2_r4.TT_06 <-> RTD Inputs Channel 4/Value
//     PlcTask Inputs/m01_rs2_r1.outlet_line_temp_error <-> RTD Inputs Channel 1/Status/Error
//     PlcTask Inputs/m01_rs2_r2.outlet_line_temp_error <-> RTD Inputs Channel 2/Status/Error
//     PlcTask Inputs/m01_rs2_r3.outlet_line_temp_error <-> RTD Inputs Channel 3/Status/Error
//     PlcTask Inputs/m01_rs2_r4.outlet_line_temp_error <-> RTD Inputs Channel 4/Status/Error
//   Phase0/Phase0 Instance <-> Device 4 (EtherCAT)/Term 1 Server Rack (EK1100)/Term 3 To DAC Mod and BOP PWR (EK1122)/Term 4 Main DAC Panel(EK1100)/Term 63 To RS2 (EK1122)/Term 64 RS2 INST Top Row (EK1100)/Term 65 (EL1008)
//     PlcTask Inputs/m01_rs2_r1.inlet_door_left_clamps_extended_ls <-> Channel 5/Input
//     PlcTask Inputs/m01_rs2_r1.inlet_door_left_closed_ls <-> Channel 2/Input
//     PlcTask Inputs/m01_rs2_r1.inlet_door_left_open_ls <-> Channel 1/Input
//     PlcTask Inputs/m01_rs2_r1.inlet_door_right_clamps_extended_ls <-> Channel 6/Input
//     PlcTask Inputs/m01_rs2_r1.inlet_door_right_closed_ls <-> Channel 4/Input
//     PlcTask Inputs/m01_rs2_r1.inlet_door_right_open_ls <-> Channel 3/Input
//     PlcTask Inputs/m01_rs2_r1.repres_valve_closed <-> Channel 7/Input
//     PlcTask Inputs/m01_rs2_r1.repres_valve_open <-> Channel 8/Input
//   Phase0/Phase0 Instance <-> Device 4 (EtherCAT)/Term 1 Server Rack (EK1100)/Term 3 To DAC Mod and BOP PWR (EK1122)/Term 4 Main DAC Panel(EK1100)/Term 63 To RS2 (EK1122)/Term 64 RS2 INST Top Row (EK1100)/Term 66 (EL1008)
//     PlcTask Inputs/m01_rs2_r1.outlet_door_left_clamps_extended_ls <-> Channel 5/Input
//     PlcTask Inputs/m01_rs2_r1.outlet_door_left_closed_ls <-> Channel 2/Input
//     PlcTask Inputs/m01_rs2_r1.outlet_door_left_open_ls <-> Channel 1/Input
//     PlcTask Inputs/m01_rs2_r1.outlet_door_right_clamps_extended_ls <-> Channel 6/Input
//     PlcTask Inputs/m01_rs2_r1.outlet_door_right_closed_ls <-> Channel 4/Input
//     PlcTask Inputs/m01_rs2_r1.outlet_door_right_open_ls <-> Channel 3/Input
//     PlcTask Inputs/m01_rs2_r3.inlet_door_left_closed_ls <-> Channel 8/Input
//     PlcTask Inputs/m01_rs2_r3.inlet_door_left_open_ls <-> Channel 7/Input
//   Phase0/Phase0 Instance <-> Device 4 (EtherCAT)/Term 1 Server Rack (EK1100)/Term 3 To DAC Mod and BOP PWR (EK1122)/Term 4 Main DAC Panel(EK1100)/Term 63 To RS2 (EK1122)/Term 64 RS2 INST Top Row (EK1100)/Term 67 (EL1008)
//     PlcTask Inputs/m01_rs2_r3.inlet_door_left_clamps_extended_ls <-> Channel 3/Input
//     PlcTask Inputs/m01_rs2_r3.inlet_door_right_clamps_extended_ls <-> Channel 4/Input
//     PlcTask Inputs/m01_rs2_r3.inlet_door_right_closed_ls <-> Channel 2/Input
//     PlcTask Inputs/m01_rs2_r3.inlet_door_right_open_ls <-> Channel 1/Input
//     PlcTask Inputs/m01_rs2_r3.outlet_door_left_closed_ls <-> Channel 8/Input
//     PlcTask Inputs/m01_rs2_r3.outlet_door_left_open_ls <-> Channel 7/Input
//     PlcTask Inputs/m01_rs2_r3.repres_valve_closed <-> Channel 5/Input
//     PlcTask Inputs/m01_rs2_r3.repres_valve_open <-> Channel 6/Input
//   Phase0/Phase0 Instance <-> Device 4 (EtherCAT)/Term 1 Server Rack (EK1100)/Term 3 To DAC Mod and BOP PWR (EK1122)/Term 4 Main DAC Panel(EK1100)/Term 63 To RS2 (EK1122)/Term 64 RS2 INST Top Row (EK1100)/Term 68 (EL1008)
//     PlcTask Inputs/m01_rs2_r2.inlet_door_left_closed_ls <-> Channel 6/Input
//     PlcTask Inputs/m01_rs2_r2.inlet_door_left_open_ls <-> Channel 5/Input
//     PlcTask Inputs/m01_rs2_r2.inlet_door_right_closed_ls <-> Channel 8/Input
//     PlcTask Inputs/m01_rs2_r2.inlet_door_right_open_ls <-> Channel 7/Input
//     PlcTask Inputs/m01_rs2_r3.outlet_door_left_clamps_extended_ls <-> Channel 3/Input
//     PlcTask Inputs/m01_rs2_r3.outlet_door_right_clamps_extended_ls <-> Channel 4/Input
//     PlcTask Inputs/m01_rs2_r3.outlet_door_right_closed_ls <-> Channel 2/Input
//     PlcTask Inputs/m01_rs2_r3.outlet_door_right_open_ls <-> Channel 1/Input
//   Phase0/Phase0 Instance <-> Device 4 (EtherCAT)/Term 1 Server Rack (EK1100)/Term 3 To DAC Mod and BOP PWR (EK1122)/Term 4 Main DAC Panel(EK1100)/Term 63 To RS2 (EK1122)/Term 64 RS2 INST Top Row (EK1100)/Term 69 (EL1008)
//     PlcTask Inputs/m01_rs2_r2.inlet_door_left_clamps_extended_ls <-> Channel 1/Input
//     PlcTask Inputs/m01_rs2_r2.inlet_door_right_clamps_extended_ls <-> Channel 2/Input
//     PlcTask Inputs/m01_rs2_r2.outlet_door_left_closed_ls <-> Channel 6/Input
//     PlcTask Inputs/m01_rs2_r2.outlet_door_left_open_ls <-> Channel 5/Input
//     PlcTask Inputs/m01_rs2_r2.outlet_door_right_closed_ls <-> Channel 8/Input
//     PlcTask Inputs/m01_rs2_r2.outlet_door_right_open_ls <-> Channel 7/Input
//     PlcTask Inputs/m01_rs2_r2.repres_valve_closed <-> Channel 3/Input
//     PlcTask Inputs/m01_rs2_r2.repres_valve_open <-> Channel 4/Input
//   Phase0/Phase0 Instance <-> Device 4 (EtherCAT)/Term 1 Server Rack (EK1100)/Term 3 To DAC Mod and BOP PWR (EK1122)/Term 4 Main DAC Panel(EK1100)/Term 63 To RS2 (EK1122)/Term 64 RS2 INST Top Row (EK1100)/Term 70 (EL1008)
//     PlcTask Inputs/m01_rs2_r2.outlet_door_left_clamps_extended_ls <-> Channel 1/Input
//     PlcTask Inputs/m01_rs2_r2.outlet_door_right_clamps_extended_ls <-> Channel 2/Input
//     PlcTask Inputs/m01_rs2_r4.inlet_door_left_clamps_extended_ls <-> Channel 7/Input
//     PlcTask Inputs/m01_rs2_r4.inlet_door_left_closed_ls <-> Channel 4/Input
//     PlcTask Inputs/m01_rs2_r4.inlet_door_left_open_ls <-> Channel 3/Input
//     PlcTask Inputs/m01_rs2_r4.inlet_door_right_clamps_extended_ls <-> Channel 8/Input
//     PlcTask Inputs/m01_rs2_r4.inlet_door_right_closed_ls <-> Channel 6/Input
//     PlcTask Inputs/m01_rs2_r4.inlet_door_right_open_ls <-> Channel 5/Input
//   Phase0/Phase0 Instance <-> Device 4 (EtherCAT)/Term 1 Server Rack (EK1100)/Term 3 To DAC Mod and BOP PWR (EK1122)/Term 4 Main DAC Panel(EK1100)/Term 63 To RS2 (EK1122)/Term 64 RS2 INST Top Row (EK1100)/Term 71 (EL1008)
//     PlcTask Inputs/m01_rs2_r4.outlet_door_left_clamps_extended_ls <-> Channel 7/Input
//     PlcTask Inputs/m01_rs2_r4.outlet_door_left_closed_ls <-> Channel 4/Input
//     PlcTask Inputs/m01_rs2_r4.outlet_door_left_open_ls <-> Channel 3/Input
//     PlcTask Inputs/m01_rs2_r4.outlet_door_right_clamps_extended_ls <-> Channel 8/Input
//     PlcTask Inputs/m01_rs2_r4.outlet_door_right_closed_ls <-> Channel 6/Input
//     PlcTask Inputs/m01_rs2_r4.outlet_door_right_open_ls <-> Channel 5/Input
//     PlcTask Inputs/m01_rs2_r4.repres_valve_closed <-> Channel 1/Input
//     PlcTask Inputs/m01_rs2_r4.repres_valve_open <-> Channel 2/Input
//   Phase0/Phase0 Instance <-> Device 4 (EtherCAT)/Term 1 Server Rack (EK1100)/Term 3 To DAC Mod and BOP PWR (EK1122)/Term 4 Main DAC Panel(EK1100)/Term 63 To RS2 (EK1122)/Term 64 RS2 INST Top Row (EK1100)/Term 72 (EL1008)
//     PlcTask Inputs/m01_rs2.cooling_valve_closed <-> Channel 5/Input
//     PlcTask Inputs/m01_rs2.cooling_valve_open <-> Channel 6/Input
//     PlcTask Inputs/m01_rs2.dead_air_valve_closed <-> Channel 1/Input
//     PlcTask Inputs/m01_rs2.dead_air_valve_open <-> Channel 2/Input
//     PlcTask Inputs/m01_rs2.purge_valve_closed <-> Channel 3/Input
//     PlcTask Inputs/m01_rs2.purge_valve_open <-> Channel 4/Input
//     PlcTask Inputs/m01_rs2.steam_header_valve_closed <-> Channel 7/Input
//     PlcTask Inputs/m01_rs2.steam_header_valve_open <-> Channel 8/Input
//   Phase0/Phase0 Instance <-> Device 4 (EtherCAT)/Term 1 Server Rack (EK1100)/Term 3 To DAC Mod and BOP PWR (EK1122)/Term 4 Main DAC Panel(EK1100)/Term 63 To RS2 (EK1122)/Term 64 RS2 INST Top Row (EK1100)/Term 73 (EL1008)
//     PlcTask Inputs/m01_rs2.condensate_lsh <-> Channel 2/Input
//     PlcTask Inputs/m01_rs2.condensate_lsl <-> Channel 1/Input
//   Phase0/Phase0 Instance <-> Device 4 (EtherCAT)/Term 1 Server Rack (EK1100)/Term 3 To DAC Mod and BOP PWR (EK1122)/Term 4 Main DAC Panel(EK1100)/Term 63 To RS2 (EK1122)/Term 64 RS2 INST Top Row (EK1100)/Term 74 (EL2008-0015)
//     PlcTask Outputs/m01_rs2_r1.AT_01_pump <-> Channel 1/Output
//     PlcTask Outputs/m01_rs2_r1.AT_03_pump <-> Channel 3/Output
//     PlcTask Outputs/m01_rs2_r1.AT_01_sol <-> Channel 2/Output
//     PlcTask Outputs/m01_rs2_r1.AT_03_sol <-> Channel 4/Output
//     PlcTask Outputs/m01_rs2_r1.XV_01_Left_Extend_Solenoid_Valve <-> Channel 6/Output
//     PlcTask Outputs/m01_rs2_r1.XV_03_Left_Extend_Solenoid_Valve <-> Channel 8/Output
//     PlcTask Outputs/m01_rs2_r1.XV_01_Right_Extend_Solenoid_Valve <-> Channel 7/Output
//     PlcTask Outputs/m01_rs2_r1.XV_02 <-> Channel 5/Output
//   Phase0/Phase0 Instance <-> Device 4 (EtherCAT)/Term 1 Server Rack (EK1100)/Term 3 To DAC Mod and BOP PWR (EK1122)/Term 4 Main DAC Panel(EK1100)/Term 63 To RS2 (EK1122)/Term 64 RS2 INST Top Row (EK1100)/Term 75 (EL2008-0015)
//     PlcTask Outputs/m01_rs2_r1.XV_03_Right_Extend_Solenoid_Valve <-> Channel 1/Output
//     PlcTask Outputs/m01_rs2_r3.XV_01_Right_Extend_Solenoid_Valve <-> Channel 8/Output
//     PlcTask Outputs/m01_rs2_r3.AT_01_pump <-> Channel 2/Output
//     PlcTask Outputs/m01_rs2_r3.AT_03_pump <-> Channel 4/Output
//     PlcTask Outputs/m01_rs2_r3.AT_01_sol <-> Channel 3/Output
//     PlcTask Outputs/m01_rs2_r3.AT_03_sol <-> Channel 5/Output
//     PlcTask Outputs/m01_rs2_r3.XV_01_Left_Extend_Solenoid_Valve <-> Channel 7/Output
//     PlcTask Outputs/m01_rs2_r3.XV_02 <-> Channel 6/Output
//   Phase0/Phase0 Instance <-> Device 4 (EtherCAT)/Term 1 Server Rack (EK1100)/Term 3 To DAC Mod and BOP PWR (EK1122)/Term 4 Main DAC Panel(EK1100)/Term 63 To RS2 (EK1122)/Term 64 RS2 INST Top Row (EK1100)/Term 76 (EL2008-0015)
//     PlcTask Outputs/m01_rs2_r2.AT_01_pump <-> Channel 3/Output
//     PlcTask Outputs/m01_rs2_r2.AT_03_pump <-> Channel 5/Output
//     PlcTask Outputs/m01_rs2_r2.AT_01_sol <-> Channel 4/Output
//     PlcTask Outputs/m01_rs2_r2.AT_03_sol <-> Channel 6/Output
//     PlcTask Outputs/m01_rs2_r2.XV_01_Left_Extend_Solenoid_Valve <-> Channel 8/Output
//     PlcTask Outputs/m01_rs2_r3.XV_03_Left_Extend_Solenoid_Valve <-> Channel 1/Output
//     PlcTask Outputs/m01_rs2_r2.XV_02 <-> Channel 7/Output
//     PlcTask Outputs/m01_rs2_r3.XV_03_Right_Extend_Solenoid_Valve <-> Channel 2/Output
//   Phase0/Phase0 Instance <-> Device 4 (EtherCAT)/Term 1 Server Rack (EK1100)/Term 3 To DAC Mod and BOP PWR (EK1122)/Term 4 Main DAC Panel(EK1100)/Term 63 To RS2 (EK1122)/Term 64 RS2 INST Top Row (EK1100)/Term 77 (EL2008-0015)
//     PlcTask Outputs/m01_rs2_r2.XV_01_Right_Extend_Solenoid_Valve <-> Channel 1/Output
//     PlcTask Outputs/m01_rs2_r2.XV_03_Right_Extend_Solenoid_Valve <-> Channel 3/Output
//     PlcTask Outputs/m01_rs2_r2.XV_03_Left_Extend_Solenoid_Valve <-> Channel 2/Output
//     PlcTask Outputs/m01_rs2_r4.AT_01_pump <-> Channel 4/Output
//     PlcTask Outputs/m01_rs2_r4.AT_03_pump <-> Channel 6/Output
//     PlcTask Outputs/m01_rs2_r4.AT_01_sol <-> Channel 5/Output
//     PlcTask Outputs/m01_rs2_r4.AT_03_sol <-> Channel 7/Output
//     PlcTask Outputs/m01_rs2_r4.XV_02 <-> Channel 8/Output
//   Phase0/Phase0 Instance <-> Device 4 (EtherCAT)/Term 1 Server Rack (EK1100)/Term 3 To DAC Mod and BOP PWR (EK1122)/Term 4 Main DAC Panel(EK1100)/Term 63 To RS2 (EK1122)/Term 64 RS2 INST Top Row (EK1100)/Term 78 (EL2008)
//     PlcTask Outputs/m01_rs2.XV_04 <-> Channel 5/Output
//     PlcTask Outputs/m01_rs2.XV_05 <-> Channel 6/Output
//     PlcTask Outputs/m01_rs2.XV_06 <-> Channel 7/Output
//     PlcTask Outputs/m01_rs2.XV_07 <-> Channel 8/Output
//     PlcTask Outputs/m01_rs2_r4.XV_01_Left_Extend_Solenoid_Valve <-> Channel 1/Output
//     PlcTask Outputs/m01_rs2_r4.XV_03_Left_Extend_Solenoid_Valve <-> Channel 3/Output
//     PlcTask Outputs/m01_rs2_r4.XV_01_Right_Extend_Solenoid_Valve <-> Channel 2/Output
//     PlcTask Outputs/m01_rs2_r4.XV_03_Right_Extend_Solenoid_Valve <-> Channel 4/Output
//   Phase0/Phase0 Instance <-> Device 4 (EtherCAT)/Term 1 Server Rack (EK1100)/Term 3 To DAC Mod and BOP PWR (EK1122)/Term 4 Main DAC Panel(EK1100)/Term 63 To RS2 (EK1122)/Term 64 RS2 INST Top Row (EK1100)/Term 79 (EL2008-0015)
//     PlcTask Outputs/m01_rs2.P_01 <-> Channel 1/Output
//   Phase0/Phase0 Instance <-> Device 4 (EtherCAT)/Term 1 Server Rack (EK1100)/Term 3 To DAC Mod and BOP PWR (EK1122)/Term 4 Main DAC Panel(EK1100)/Term 63 To RS2 (EK1122)/Term 64 RS2 INST Top Row (EK1100)/Term 80 (EL2008-0015)
//     PlcTask Outputs/m01_rs2_r1.XV_01_Left_Retract_Solenoid_Valve <-> Channel 1/Output
//     PlcTask Outputs/m01_rs2_r1.XV_03_Left_Retract_Solenoid_Valve <-> Channel 3/Output
//     PlcTask Outputs/m01_rs2_r3.XV_01_Left_Retract_Solenoid_Valve <-> Channel 5/Output
//     PlcTask Outputs/m01_rs2_r3.XV_03_Left_Retract_Solenoid_Valve <-> Channel 7/Output
//     PlcTask Outputs/m01_rs2_r1.XV_01_Right_Retract_Solenoid_Valve <-> Channel 2/Output
//     PlcTask Outputs/m01_rs2_r1.XV_03_Right_Retract_Solenoid_Valve <-> Channel 4/Output
//     PlcTask Outputs/m01_rs2_r3.XV_01_Right_Retract_Solenoid_Valve <-> Channel 6/Output
//     PlcTask Outputs/m01_rs2_r3.XV_03_Right_Retract_Solenoid_Valve <-> Channel 8/Output
//   Phase0/Phase0 Instance <-> Device 4 (EtherCAT)/Term 1 Server Rack (EK1100)/Term 3 To DAC Mod and BOP PWR (EK1122)/Term 4 Main DAC Panel(EK1100)/Term 63 To RS2 (EK1122)/Term 64 RS2 INST Top Row (EK1100)/Term 81 (EL2008-0015)
//     PlcTask Outputs/m01_rs2_r2.XV_01_Left_Retract_Solenoid_Valve <-> Channel 1/Output
//     PlcTask Outputs/m01_rs2_r2.XV_03_Left_Retract_Solenoid_Valve <-> Channel 3/Output
//     PlcTask Outputs/m01_rs2_r4.XV_01_Left_Retract_Solenoid_Valve <-> Channel 5/Output
//     PlcTask Outputs/m01_rs2_r4.XV_03_Left_Retract_Solenoid_Valve <-> Channel 7/Output
//     PlcTask Outputs/m01_rs2_r2.XV_01_Right_Retract_Solenoid_Valve <-> Channel 2/Output
//     PlcTask Outputs/m01_rs2_r2.XV_03_Right_Retract_Solenoid_Valve <-> Channel 4/Output
//     PlcTask Outputs/m01_rs2_r4.XV_01_Right_Retract_Solenoid_Valve <-> Channel 6/Output
//     PlcTask Outputs/m01_rs2_r4.XV_03_Right_Retract_Solenoid_Valve <-> Channel 8/Output
//   Phase0/Phase0 Instance <-> Device 4 (EtherCAT)/Term 1 Server Rack (EK1100)/Term 3 To DAC Mod and BOP PWR (EK1122)/Term 4 Main DAC Panel(EK1100)/Term 63 To RS2 (EK1122)/Term 64 RS2 INST Top Row (EK1100)/Term 82 (EL3058)
//     PlcTask Inputs/m01_rs2_r1.AT_01 <-> AI Standard Channel 1/Value
//     PlcTask Inputs/m01_rs2_r1.AT_02 <-> AI Standard Channel 2/Value
//     PlcTask Inputs/m01_rs2_r1.AT_03 <-> AI Standard Channel 3/Value
//     PlcTask Inputs/m01_rs2_r1.AT_04 <-> AI Standard Channel 4/Value
//     PlcTask Inputs/m01_rs2_r1.FT_01 <-> AI Standard Channel 5/Value
//     PlcTask Inputs/m01_rs2_r1.PDT_01 <-> AI Standard Channel 6/Value
//     PlcTask Inputs/m01_rs2_r1.PDT_02 <-> AI Standard Channel 7/Value
//     PlcTask Inputs/m01_rs2_r1.PDT_03 <-> AI Standard Channel 8/Value
//     PlcTask Inputs/m01_rs2_r1.air_flow_error <-> AI Standard Channel 5/Status/Error
//     PlcTask Inputs/m01_rs2_r1.fan_diff_pres_error <-> AI Standard Channel 8/Status/Error
//     PlcTask Inputs/m01_rs2_r1.filter_diff_pres_error <-> AI Standard Channel 6/Status/Error
//     PlcTask Inputs/m01_rs2_r1.inlet_co2_error <-> AI Standard Channel 1/Status/Error
//     PlcTask Inputs/m01_rs2_r1.inlet_h2o_error <-> AI Standard Channel 2/Status/Error
//     PlcTask Inputs/m01_rs2_r1.outlet_co2_error <-> AI Standard Channel 3/Status/Error
//     PlcTask Inputs/m01_rs2_r1.outlet_h2o_error <-> AI Standard Channel 4/Status/Error
//     PlcTask Inputs/m01_rs2_r1.sorbent_diff_pres_error <-> AI Standard Channel 7/Status/Error
//   Phase0/Phase0 Instance <-> Device 4 (EtherCAT)/Term 1 Server Rack (EK1100)/Term 3 To DAC Mod and BOP PWR (EK1122)/Term 4 Main DAC Panel(EK1100)/Term 63 To RS2 (EK1122)/Term 64 RS2 INST Top Row (EK1100)/Term 84 (EL3058)
//     PlcTask Inputs/m01_rs2_r1.PT_01 <-> AI Standard Channel 1/Value
//     PlcTask Inputs/m01_rs2_r1.reactor_pres_error <-> AI Standard Channel 1/Status/Error
//     PlcTask Inputs/m01_rs2_r2.air_flow_error <-> AI Standard Channel 6/Status/Error
//     PlcTask Inputs/m01_rs2_r2.filter_diff_pres_error <-> AI Standard Channel 7/Status/Error
//     PlcTask Inputs/m01_rs2_r2.inlet_co2_error <-> AI Standard Channel 2/Status/Error
//     PlcTask Inputs/m01_rs2_r2.inlet_h2o_error <-> AI Standard Channel 3/Status/Error
//     PlcTask Inputs/m01_rs2_r2.outlet_co2_error <-> AI Standard Channel 4/Status/Error
//     PlcTask Inputs/m01_rs2_r2.outlet_h2o_error <-> AI Standard Channel 5/Status/Error
//     PlcTask Inputs/m01_rs2_r2.sorbent_diff_pres_error <-> AI Standard Channel 8/Status/Error
//     PlcTask Inputs/m01_rs2_r3.AT_01 <-> AI Standard Channel 2/Value
//     PlcTask Inputs/m01_rs2_r3.AT_02 <-> AI Standard Channel 3/Value
//     PlcTask Inputs/m01_rs2_r3.AT_03 <-> AI Standard Channel 4/Value
//     PlcTask Inputs/m01_rs2_r3.AT_04 <-> AI Standard Channel 5/Value
//     PlcTask Inputs/m01_rs2_r3.FT_01 <-> AI Standard Channel 6/Value
//     PlcTask Inputs/m01_rs2_r3.PDT_01 <-> AI Standard Channel 7/Value
//     PlcTask Inputs/m01_rs2_r3.PDT_02 <-> AI Standard Channel 8/Value
//   Phase0/Phase0 Instance <-> Device 4 (EtherCAT)/Term 1 Server Rack (EK1100)/Term 3 To DAC Mod and BOP PWR (EK1122)/Term 4 Main DAC Panel(EK1100)/Term 63 To RS2 (EK1122)/Term 64 RS2 INST Top Row (EK1100)/Term 85 (EL3058)
//     PlcTask Inputs/m01_rs2_r2.AT_01 <-> AI Standard Channel 3/Value
//     PlcTask Inputs/m01_rs2_r2.AT_02 <-> AI Standard Channel 4/Value
//     PlcTask Inputs/m01_rs2_r2.AT_03 <-> AI Standard Channel 5/Value
//     PlcTask Inputs/m01_rs2_r2.AT_04 <-> AI Standard Channel 6/Value
//     PlcTask Inputs/m01_rs2_r2.FT_01 <-> AI Standard Channel 7/Value
//     PlcTask Inputs/m01_rs2_r2.PDT_01 <-> AI Standard Channel 8/Value
//     PlcTask Inputs/m01_rs2_r3.PDT_03 <-> AI Standard Channel 1/Value
//     PlcTask Inputs/m01_rs2_r2.fan_diff_pres_error <-> AI Standard Channel 1/Status/Error
//     PlcTask Inputs/m01_rs2_r2.reactor_pres_error <-> AI Standard Channel 2/Status/Error
//     PlcTask Inputs/m01_rs2_r3.PT_01 <-> AI Standard Channel 2/Value
//     PlcTask Inputs/m01_rs2_r3.air_flow_error <-> AI Standard Channel 7/Status/Error
//     PlcTask Inputs/m01_rs2_r3.filter_diff_pres_error <-> AI Standard Channel 8/Status/Error
//     PlcTask Inputs/m01_rs2_r3.inlet_co2_error <-> AI Standard Channel 3/Status/Error
//     PlcTask Inputs/m01_rs2_r3.inlet_h2o_error <-> AI Standard Channel 4/Status/Error
//     PlcTask Inputs/m01_rs2_r3.outlet_co2_error <-> AI Standard Channel 5/Status/Error
//     PlcTask Inputs/m01_rs2_r3.outlet_h2o_error <-> AI Standard Channel 6/Status/Error
//   Phase0/Phase0 Instance <-> Device 4 (EtherCAT)/Term 1 Server Rack (EK1100)/Term 3 To DAC Mod and BOP PWR (EK1122)/Term 4 Main DAC Panel(EK1100)/Term 63 To RS2 (EK1122)/Term 64 RS2 INST Top Row (EK1100)/Term 86 (EL3058)
//     PlcTask Inputs/m01_rs2_r2.PDT_02 <-> AI Standard Channel 1/Value
//     PlcTask Inputs/m01_rs2_r2.PDT_03 <-> AI Standard Channel 2/Value
//     PlcTask Inputs/m01_rs2_r2.PT_01 <-> AI Standard Channel 3/Value
//     PlcTask Inputs/m01_rs2_r3.fan_diff_pres_error <-> AI Standard Channel 2/Status/Error
//     PlcTask Inputs/m01_rs2_r3.reactor_pres_error <-> AI Standard Channel 3/Status/Error
//     PlcTask Inputs/m01_rs2_r3.sorbent_diff_pres_error <-> AI Standard Channel 1/Status/Error
//     PlcTask Inputs/m01_rs2_r4.AT_01 <-> AI Standard Channel 4/Value
//     PlcTask Inputs/m01_rs2_r4.AT_02 <-> AI Standard Channel 5/Value
//     PlcTask Inputs/m01_rs2_r4.AT_03 <-> AI Standard Channel 6/Value
//     PlcTask Inputs/m01_rs2_r4.AT_04 <-> AI Standard Channel 7/Value
//     PlcTask Inputs/m01_rs2_r4.FT_01 <-> AI Standard Channel 8/Value
//     PlcTask Inputs/m01_rs2_r4.air_flow_error <-> AI Standard Channel 8/Status/Error
//     PlcTask Inputs/m01_rs2_r4.inlet_co2_error <-> AI Standard Channel 4/Status/Error
//     PlcTask Inputs/m01_rs2_r4.inlet_h2o_error <-> AI Standard Channel 5/Status/Error
//     PlcTask Inputs/m01_rs2_r4.outlet_co2_error <-> AI Standard Channel 6/Status/Error
//     PlcTask Inputs/m01_rs2_r4.outlet_h2o_error <-> AI Standard Channel 7/Status/Error
//   Phase0/Phase0 Instance <-> Device 4 (EtherCAT)/Term 1 Server Rack (EK1100)/Term 3 To DAC Mod and BOP PWR (EK1122)/Term 4 Main DAC Panel(EK1100)/Term 63 To RS2 (EK1122)/Term 64 RS2 INST Top Row (EK1100)/Term 87 (EL3058)
//     PlcTask Inputs/m01_rs2.PCV_01_position <-> AI Standard Channel 5/Value
//     PlcTask Inputs/m01_rs2.steam_control_valve_position_error <-> AI Standard Channel 5/Status/Error
//     PlcTask Inputs/m01_rs2_r4.PDT_01 <-> AI Standard Channel 1/Value
//     PlcTask Inputs/m01_rs2_r4.PDT_02 <-> AI Standard Channel 2/Value
//     PlcTask Inputs/m01_rs2_r4.PDT_03 <-> AI Standard Channel 3/Value
//     PlcTask Inputs/m01_rs2_r4.PT_01 <-> AI Standard Channel 4/Value
//     PlcTask Inputs/m01_rs2_r4.fan_diff_pres_error <-> AI Standard Channel 3/Status/Error
//     PlcTask Inputs/m01_rs2_r4.filter_diff_pres_error <-> AI Standard Channel 1/Status/Error
//     PlcTask Inputs/m01_rs2_r4.reactor_pres_error <-> AI Standard Channel 4/Status/Error
//     PlcTask Inputs/m01_rs2_r4.sorbent_diff_pres_error <-> AI Standard Channel 2/Status/Error
//   Phase0/Phase0 Instance <-> Device 4 (EtherCAT)/Term 1 Server Rack (EK1100)/Term 3 To DAC Mod and BOP PWR (EK1122)/Term 4 Main DAC Panel(EK1100)/Term 63 To RS2 (EK1122)/Term 64 RS2 INST Top Row (EK1100)/Term 88 (EL4122)
//     PlcTask Outputs/m01_rs2.PCV_01 <-> Channel 1/Output
//   Phase0/Phase0 Instance <-> Device 4 (EtherCAT)/Term 1 Server Rack (EK1100)/Term 3 To DAC Mod and BOP PWR (EK1122)/Term 4 Main DAC Panel(EK1100)/Term 63 To RS2 (EK1122)/Term 64 RS2 INST Top Row (EK1100)/Term 89 (EL3318)
//     PlcTask Inputs/m01_rs2_r1._01_TT_01 <-> TC Channel 1/Value
//     PlcTask Inputs/m01_rs2_r1._01_TT_03 <-> TC Channel 2/Value
//     PlcTask Inputs/m01_rs2_r1._02_TT_01 <-> TC Channel 3/Value
//     PlcTask Inputs/m01_rs2_r1._02_TT_03 <-> TC Channel 4/Value
//     PlcTask Inputs/m01_rs2_r1._03_TT_01 <-> TC Channel 5/Value
//     PlcTask Inputs/m01_rs2_r1._03_TT_03 <-> TC Channel 6/Value
//     PlcTask Inputs/m01_rs2_r1._04_TT_01 <-> TC Channel 7/Value
//     PlcTask Inputs/m01_rs2_r1._04_TT_03 <-> TC Channel 8/Value
//     PlcTask Inputs/m01_rs2_r1._01_TT_01_Error <-> TC Channel 1/Status/Error
//     PlcTask Inputs/m01_rs2_r1._01_TT_03_Error <-> TC Channel 2/Status/Error
//     PlcTask Inputs/m01_rs2_r1._02_TT_01_Error <-> TC Channel 3/Status/Error
//     PlcTask Inputs/m01_rs2_r1._02_TT_03_Error <-> TC Channel 4/Status/Error
//     PlcTask Inputs/m01_rs2_r1._03_TT_01_Error <-> TC Channel 5/Status/Error
//     PlcTask Inputs/m01_rs2_r1._03_TT_03_Error <-> TC Channel 6/Status/Error
//     PlcTask Inputs/m01_rs2_r1._04_TT_01_Error <-> TC Channel 7/Status/Error
//     PlcTask Inputs/m01_rs2_r1._04_TT_03_Error <-> TC Channel 8/Status/Error
//   Phase0/Phase0 Instance <-> Device 4 (EtherCAT)/Term 1 Server Rack (EK1100)/Term 3 To DAC Mod and BOP PWR (EK1122)/Term 4 Main DAC Panel(EK1100)/Term 63 To RS2 (EK1122)/Term 64 RS2 INST Top Row (EK1100)/Term 90 (EL3318)
//     PlcTask Inputs/m01_rs2_r1._05_TT_01 <-> TC Channel 1/Value
//     PlcTask Inputs/m01_rs2_r1._05_TT_03 <-> TC Channel 2/Value
//     PlcTask Inputs/m01_rs2_r1._06_TT_01 <-> TC Channel 3/Value
//     PlcTask Inputs/m01_rs2_r1._06_TT_03 <-> TC Channel 4/Value
//     PlcTask Inputs/m01_rs2_r1._07_TT_01 <-> TC Channel 5/Value
//     PlcTask Inputs/m01_rs2_r1._07_TT_03 <-> TC Channel 6/Value
//     PlcTask Inputs/m01_rs2_r1._08_TT_01 <-> TC Channel 7/Value
//     PlcTask Inputs/m01_rs2_r1._08_TT_03 <-> TC Channel 8/Value
//     PlcTask Inputs/m01_rs2_r1._05_TT_01_Error <-> TC Channel 1/Status/Error
//     PlcTask Inputs/m01_rs2_r1._05_TT_03_Error <-> TC Channel 2/Status/Error
//     PlcTask Inputs/m01_rs2_r1._06_TT_01_Error <-> TC Channel 3/Status/Error
//     PlcTask Inputs/m01_rs2_r1._06_TT_03_Error <-> TC Channel 4/Status/Error
//     PlcTask Inputs/m01_rs2_r1._07_TT_01_Error <-> TC Channel 5/Status/Error
//     PlcTask Inputs/m01_rs2_r1._07_TT_03_Error <-> TC Channel 6/Status/Error
//     PlcTask Inputs/m01_rs2_r1._08_TT_01_Error <-> TC Channel 7/Status/Error
//     PlcTask Inputs/m01_rs2_r1._08_TT_03_Error <-> TC Channel 8/Status/Error
//   Phase0/Phase0 Instance <-> Device 4 (EtherCAT)/Term 1 Server Rack (EK1100)/Term 3 To DAC Mod and BOP PWR (EK1122)/Term 4 Main DAC Panel(EK1100)/Term 63 To RS2 (EK1122)/Term 64 RS2 INST Top Row (EK1100)/Term 91 (EL3318)
//     PlcTask Inputs/m01_rs2_r1._09_TT_01 <-> TC Channel 1/Value
//     PlcTask Inputs/m01_rs2_r1._09_TT_03 <-> TC Channel 2/Value
//     PlcTask Inputs/m01_rs2_r1._10_TT_01 <-> TC Channel 3/Value
//     PlcTask Inputs/m01_rs2_r1._10_TT_03 <-> TC Channel 4/Value
//     PlcTask Inputs/m01_rs2_r1._11_TT_01 <-> TC Channel 5/Value
//     PlcTask Inputs/m01_rs2_r1._11_TT_03 <-> TC Channel 6/Value
//     PlcTask Inputs/m01_rs2_r1._12_TT_01 <-> TC Channel 7/Value
//     PlcTask Inputs/m01_rs2_r1._12_TT_03 <-> TC Channel 8/Value
//     PlcTask Inputs/m01_rs2_r1._09_TT_01_Error <-> TC Channel 1/Status/Error
//     PlcTask Inputs/m01_rs2_r1._09_TT_03_Error <-> TC Channel 2/Status/Error
//     PlcTask Inputs/m01_rs2_r1._10_TT_01_Error <-> TC Channel 3/Status/Error
//     PlcTask Inputs/m01_rs2_r1._10_TT_03_Error <-> TC Channel 4/Status/Error
//     PlcTask Inputs/m01_rs2_r1._11_TT_01_Error <-> TC Channel 5/Status/Error
//     PlcTask Inputs/m01_rs2_r1._11_TT_03_Error <-> TC Channel 6/Status/Error
//     PlcTask Inputs/m01_rs2_r1._12_TT_01_Error <-> TC Channel 7/Status/Error
//     PlcTask Inputs/m01_rs2_r1._12_TT_03_Error <-> TC Channel 8/Status/Error
//   Phase0/Phase0 Instance <-> Device 4 (EtherCAT)/Term 1 Server Rack (EK1100)/Term 3 To DAC Mod and BOP PWR (EK1122)/Term 4 Main DAC Panel(EK1100)/Term 63 To RS2 (EK1122)/Term 64 RS2 INST Top Row (EK1100)/Term 92 (EL3318)
//     PlcTask Inputs/m01_rs2_r3._01_TT_01 <-> TC Channel 1/Value
//     PlcTask Inputs/m01_rs2_r3._01_TT_03 <-> TC Channel 2/Value
//     PlcTask Inputs/m01_rs2_r3._02_TT_01 <-> TC Channel 3/Value
//     PlcTask Inputs/m01_rs2_r3._02_TT_03 <-> TC Channel 4/Value
//     PlcTask Inputs/m01_rs2_r3._03_TT_01 <-> TC Channel 5/Value
//     PlcTask Inputs/m01_rs2_r3._03_TT_03 <-> TC Channel 6/Value
//     PlcTask Inputs/m01_rs2_r3._04_TT_01 <-> TC Channel 7/Value
//     PlcTask Inputs/m01_rs2_r3._04_TT_03 <-> TC Channel 8/Value
//     PlcTask Inputs/m01_rs2_r3._01_TT_01_Error <-> TC Channel 1/Status/Error
//     PlcTask Inputs/m01_rs2_r3._01_TT_03_Error <-> TC Channel 2/Status/Error
//     PlcTask Inputs/m01_rs2_r3._02_TT_01_Error <-> TC Channel 3/Status/Error
//     PlcTask Inputs/m01_rs2_r3._02_TT_03_Error <-> TC Channel 4/Status/Error
//     PlcTask Inputs/m01_rs2_r3._03_TT_01_Error <-> TC Channel 5/Status/Error
//     PlcTask Inputs/m01_rs2_r3._03_TT_03_Error <-> TC Channel 6/Status/Error
//     PlcTask Inputs/m01_rs2_r3._04_TT_01_Error <-> TC Channel 7/Status/Error
//     PlcTask Inputs/m01_rs2_r3._04_TT_03_Error <-> TC Channel 8/Status/Error
//   Phase0/Phase0 Instance <-> Device 4 (EtherCAT)/Term 1 Server Rack (EK1100)/Term 3 To DAC Mod and BOP PWR (EK1122)/Term 4 Main DAC Panel(EK1100)/Term 63 To RS2 (EK1122)/Term 64 RS2 INST Top Row (EK1100)/Term 93 (EL3318)
//     PlcTask Inputs/m01_rs2_r3._05_TT_01 <-> TC Channel 1/Value
//     PlcTask Inputs/m01_rs2_r3._05_TT_03 <-> TC Channel 2/Value
//     PlcTask Inputs/m01_rs2_r3._06_TT_01 <-> TC Channel 3/Value
//     PlcTask Inputs/m01_rs2_r3._06_TT_03 <-> TC Channel 4/Value
//     PlcTask Inputs/m01_rs2_r3._07_TT_01 <-> TC Channel 5/Value
//     PlcTask Inputs/m01_rs2_r3._07_TT_03 <-> TC Channel 6/Value
//     PlcTask Inputs/m01_rs2_r3._08_TT_01 <-> TC Channel 7/Value
//     PlcTask Inputs/m01_rs2_r3._08_TT_03 <-> TC Channel 8/Value
//     PlcTask Inputs/m01_rs2_r3._05_TT_01_Error <-> TC Channel 1/Status/Error
//     PlcTask Inputs/m01_rs2_r3._05_TT_03_Error <-> TC Channel 2/Status/Error
//     PlcTask Inputs/m01_rs2_r3._06_TT_01_Error <-> TC Channel 3/Status/Error
//     PlcTask Inputs/m01_rs2_r3._06_TT_03_Error <-> TC Channel 4/Status/Error
//     PlcTask Inputs/m01_rs2_r3._07_TT_01_Error <-> TC Channel 5/Status/Error
//     PlcTask Inputs/m01_rs2_r3._07_TT_03_Error <-> TC Channel 6/Status/Error
//     PlcTask Inputs/m01_rs2_r3._08_TT_01_Error <-> TC Channel 7/Status/Error
//     PlcTask Inputs/m01_rs2_r3._08_TT_03_Error <-> TC Channel 8/Status/Error
//   Phase0/Phase0 Instance <-> Device 4 (EtherCAT)/Term 1 Server Rack (EK1100)/Term 3 To DAC Mod and BOP PWR (EK1122)/Term 4 Main DAC Panel(EK1100)/Term 63 To RS2 (EK1122)/Term 64 RS2 INST Top Row (EK1100)/Term 94 (EL3318)
//     PlcTask Inputs/m01_rs2_r3._09_TT_01 <-> TC Channel 1/Value
//     PlcTask Inputs/m01_rs2_r3._09_TT_03 <-> TC Channel 2/Value
//     PlcTask Inputs/m01_rs2_r3._10_TT_01 <-> TC Channel 3/Value
//     PlcTask Inputs/m01_rs2_r3._10_TT_03 <-> TC Channel 4/Value
//     PlcTask Inputs/m01_rs2_r3._11_TT_01 <-> TC Channel 5/Value
//     PlcTask Inputs/m01_rs2_r3._11_TT_03 <-> TC Channel 6/Value
//     PlcTask Inputs/m01_rs2_r3._12_TT_01 <-> TC Channel 7/Value
//     PlcTask Inputs/m01_rs2_r3._12_TT_03 <-> TC Channel 8/Value
//     PlcTask Inputs/m01_rs2_r3._09_TT_01_Error <-> TC Channel 1/Status/Error
//     PlcTask Inputs/m01_rs2_r3._09_TT_03_Error <-> TC Channel 2/Status/Error
//     PlcTask Inputs/m01_rs2_r3._10_TT_01_Error <-> TC Channel 3/Status/Error
//     PlcTask Inputs/m01_rs2_r3._10_TT_03_Error <-> TC Channel 4/Status/Error
//     PlcTask Inputs/m01_rs2_r3._11_TT_01_Error <-> TC Channel 5/Status/Error
//     PlcTask Inputs/m01_rs2_r3._11_TT_03_Error <-> TC Channel 6/Status/Error
//     PlcTask Inputs/m01_rs2_r3._12_TT_01_Error <-> TC Channel 7/Status/Error
//     PlcTask Inputs/m01_rs2_r3._12_TT_03_Error <-> TC Channel 8/Status/Error
//   Phase0/Phase0 Instance <-> Device 4 (EtherCAT)/Term 1 Server Rack (EK1100)/Term 3 To DAC Mod and BOP PWR (EK1122)/Term 4 Main DAC Panel(EK1100)/Term 63 To RS2 (EK1122)/Term 64 RS2 INST Top Row (EK1100)/Term 96 (EL3318)
//     PlcTask Inputs/m01_rs2_r2._01_TT_01 <-> TC Channel 1/Value
//     PlcTask Inputs/m01_rs2_r2._01_TT_03 <-> TC Channel 2/Value
//     PlcTask Inputs/m01_rs2_r2._02_TT_01 <-> TC Channel 3/Value
//     PlcTask Inputs/m01_rs2_r2._02_TT_03 <-> TC Channel 4/Value
//     PlcTask Inputs/m01_rs2_r2._03_TT_01 <-> TC Channel 5/Value
//     PlcTask Inputs/m01_rs2_r2._03_TT_03 <-> TC Channel 6/Value
//     PlcTask Inputs/m01_rs2_r2._04_TT_01 <-> TC Channel 7/Value
//     PlcTask Inputs/m01_rs2_r2._04_TT_03 <-> TC Channel 8/Value
//     PlcTask Inputs/m01_rs2_r2._01_TT_01_Error <-> TC Channel 1/Status/Error
//     PlcTask Inputs/m01_rs2_r2._01_TT_03_Error <-> TC Channel 2/Status/Error
//     PlcTask Inputs/m01_rs2_r2._02_TT_01_Error <-> TC Channel 3/Status/Error
//     PlcTask Inputs/m01_rs2_r2._02_TT_03_Error <-> TC Channel 4/Status/Error
//     PlcTask Inputs/m01_rs2_r2._03_TT_01_Error <-> TC Channel 5/Status/Error
//     PlcTask Inputs/m01_rs2_r2._03_TT_03_Error <-> TC Channel 6/Status/Error
//     PlcTask Inputs/m01_rs2_r2._04_TT_01_Error <-> TC Channel 7/Status/Error
//     PlcTask Inputs/m01_rs2_r2._04_TT_03_Error <-> TC Channel 8/Status/Error
//   Phase0/Phase0 Instance <-> Device 4 (EtherCAT)/Term 1 Server Rack (EK1100)/Term 3 To DAC Mod and BOP PWR (EK1122)/Term 4 Main DAC Panel(EK1100)/Term 63 To RS2 (EK1122)/Term 64 RS2 INST Top Row (EK1100)/Term 97 (EL3318)
//     PlcTask Inputs/m01_rs2_r2._05_TT_01 <-> TC Channel 1/Value
//     PlcTask Inputs/m01_rs2_r2._05_TT_03 <-> TC Channel 2/Value
//     PlcTask Inputs/m01_rs2_r2._06_TT_01 <-> TC Channel 3/Value
//     PlcTask Inputs/m01_rs2_r2._06_TT_03 <-> TC Channel 4/Value
//     PlcTask Inputs/m01_rs2_r2._07_TT_01 <-> TC Channel 5/Value
//     PlcTask Inputs/m01_rs2_r2._07_TT_03 <-> TC Channel 6/Value
//     PlcTask Inputs/m01_rs2_r2._08_TT_01 <-> TC Channel 7/Value
//     PlcTask Inputs/m01_rs2_r2._08_TT_03 <-> TC Channel 8/Value
//     PlcTask Inputs/m01_rs2_r2._05_TT_01_Error <-> TC Channel 1/Status/Error
//     PlcTask Inputs/m01_rs2_r2._05_TT_03_Error <-> TC Channel 2/Status/Error
//     PlcTask Inputs/m01_rs2_r2._06_TT_01_Error <-> TC Channel 3/Status/Error
//     PlcTask Inputs/m01_rs2_r2._06_TT_03_Error <-> TC Channel 4/Status/Error
//     PlcTask Inputs/m01_rs2_r2._07_TT_01_Error <-> TC Channel 5/Status/Error
//     PlcTask Inputs/m01_rs2_r2._07_TT_03_Error <-> TC Channel 6/Status/Error
//     PlcTask Inputs/m01_rs2_r2._08_TT_01_Error <-> TC Channel 7/Status/Error
//     PlcTask Inputs/m01_rs2_r2._08_TT_03_Error <-> TC Channel 8/Status/Error
//   Phase0/Phase0 Instance <-> Device 4 (EtherCAT)/Term 1 Server Rack (EK1100)/Term 3 To DAC Mod and BOP PWR (EK1122)/Term 4 Main DAC Panel(EK1100)/Term 63 To RS2 (EK1122)/Term 64 RS2 INST Top Row (EK1100)/Term 98 (EL3318)
//     PlcTask Inputs/m01_rs2_r2._09_TT_01 <-> TC Channel 1/Value
//     PlcTask Inputs/m01_rs2_r2._09_TT_03 <-> TC Channel 2/Value
//     PlcTask Inputs/m01_rs2_r2._10_TT_01 <-> TC Channel 3/Value
//     PlcTask Inputs/m01_rs2_r2._10_TT_03 <-> TC Channel 4/Value
//     PlcTask Inputs/m01_rs2_r2._11_TT_01 <-> TC Channel 5/Value
//     PlcTask Inputs/m01_rs2_r2._11_TT_03 <-> TC Channel 6/Value
//     PlcTask Inputs/m01_rs2_r2._12_TT_01 <-> TC Channel 7/Value
//     PlcTask Inputs/m01_rs2_r2._12_TT_03 <-> TC Channel 8/Value
//     PlcTask Inputs/m01_rs2_r2._09_TT_01_Error <-> TC Channel 1/Status/Error
//     PlcTask Inputs/m01_rs2_r2._09_TT_03_Error <-> TC Channel 2/Status/Error
//     PlcTask Inputs/m01_rs2_r2._10_TT_01_Error <-> TC Channel 3/Status/Error
//     PlcTask Inputs/m01_rs2_r2._10_TT_03_Error <-> TC Channel 4/Status/Error
//     PlcTask Inputs/m01_rs2_r2._11_TT_01_Error <-> TC Channel 5/Status/Error
//     PlcTask Inputs/m01_rs2_r2._11_TT_03_Error <-> TC Channel 6/Status/Error
//     PlcTask Inputs/m01_rs2_r2._12_TT_01_Error <-> TC Channel 7/Status/Error
//     PlcTask Inputs/m01_rs2_r2._12_TT_03_Error <-> TC Channel 8/Status/Error
//   Phase0/Phase0 Instance <-> Device 4 (EtherCAT)/Term 1 Server Rack (EK1100)/Term 3 To DAC Mod and BOP PWR (EK1122)/Term 4 Main DAC Panel(EK1100)/Term 63 To RS2 (EK1122)/Term 64 RS2 INST Top Row (EK1100)/Term 99 (EL3318)
//     PlcTask Inputs/m01_rs2_r4._01_TT_01 <-> TC Channel 1/Value
//     PlcTask Inputs/m01_rs2_r4._01_TT_03 <-> TC Channel 2/Value
//     PlcTask Inputs/m01_rs2_r4._02_TT_01 <-> TC Channel 3/Value
//     PlcTask Inputs/m01_rs2_r4._02_TT_03 <-> TC Channel 4/Value
//     PlcTask Inputs/m01_rs2_r4._03_TT_01 <-> TC Channel 5/Value
//     PlcTask Inputs/m01_rs2_r4._03_TT_03 <-> TC Channel 6/Value
//     PlcTask Inputs/m01_rs2_r4._04_TT_01 <-> TC Channel 7/Value
//     PlcTask Inputs/m01_rs2_r4._04_TT_03 <-> TC Channel 8/Value
//     PlcTask Inputs/m01_rs2_r4._01_TT_01_Error <-> TC Channel 1/Status/Error
//     PlcTask Inputs/m01_rs2_r4._01_TT_03_Error <-> TC Channel 2/Status/Error
//     PlcTask Inputs/m01_rs2_r4._02_TT_01_Error <-> TC Channel 3/Status/Error
//     PlcTask Inputs/m01_rs2_r4._02_TT_03_Error <-> TC Channel 4/Status/Error
//     PlcTask Inputs/m01_rs2_r4._03_TT_01_Error <-> TC Channel 5/Status/Error
//     PlcTask Inputs/m01_rs2_r4._03_TT_03_Error <-> TC Channel 6/Status/Error
//     PlcTask Inputs/m01_rs2_r4._04_TT_01_Error <-> TC Channel 7/Status/Error
//     PlcTask Inputs/m01_rs2_r4._04_TT_03_Error <-> TC Channel 8/Status/Error
//   Phase0/Phase0 Instance <-> Device 4 (EtherCAT)/Term 1 Server Rack (EK1100)/Term 3 To DAC Mod and BOP PWR (EK1122)/Term 4 Main DAC Panel(EK1100)/Term 7 (EL2008)
//     PlcTask Outputs/m01.P_02 <-> Channel 4/Output
//     PlcTask Outputs/m01_rs1.PWR_01 <-> Channel 2/Output
//     PlcTask Outputs/m01_rs2.PWR_01 <-> Channel 3/Output
//     PlcTask Outputs/m01_rs3.PWR_01 <-> Channel 1/Output
//   Phase0/Phase0 Instance <-> Device 4 (EtherCAT)/Term 1 Server Rack (EK1100)/Term 3 To DAC Mod and BOP PWR (EK1122)/Term 4 Main DAC Panel(EK1100)/Term 8 (EL3058)
//     PlcTask Inputs/m01.FT_02 <-> AI Standard Channel 2/Value
//     PlcTask Inputs/m01.IT_01 <-> AI Standard Channel 6/Value
//     PlcTask Inputs/m01.IT_02 <-> AI Standard Channel 7/Value
//     PlcTask Inputs/m01.IT_03 <-> AI Standard Channel 8/Value
//     PlcTask Inputs/m01.PT_02 <-> AI Standard Channel 1/Value
//     PlcTask Inputs/m01.VT_01 <-> AI Standard Channel 3/Value
//     PlcTask Inputs/m01.VT_02 <-> AI Standard Channel 4/Value
//     PlcTask Inputs/m01.VT_03 <-> AI Standard Channel 5/Value
//     PlcTask Inputs/m01.condensate_flow_error <-> AI Standard Channel 2/Status/Error
//     PlcTask Inputs/m01.l1_current_error <-> AI Standard Channel 6/Status/Error
//     PlcTask Inputs/m01.l2_current_error <-> AI Standard Channel 7/Status/Error
//     PlcTask Inputs/m01.l3_current_error <-> AI Standard Channel 8/Status/Error
//     PlcTask Inputs/m01.l1_volatge_error <-> AI Standard Channel 3/Status/Error
//     PlcTask Inputs/m01.l2_volatge_error <-> AI Standard Channel 4/Status/Error
//     PlcTask Inputs/m01.l3_volatge_error <-> AI Standard Channel 5/Status/Error
//     PlcTask Inputs/m01.steam_manifold_line_pres_error <-> AI Standard Channel 1/Status/Error
//   Phase0/Phase0 Instance <-> Device 4 (EtherCAT)/Term 1 Server Rack (EK1100)/Term 3 To DAC Mod and BOP PWR (EK1122)/Term 4 Main DAC Panel(EK1100)/Term 9 (EL3214)
//     PlcTask Inputs/m01.TT_10 <-> RTD Inputs Channel 1/Value
//     PlcTask Inputs/m01.TT_11 <-> RTD Inputs Channel 2/Value
//     PlcTask Inputs/m01.TT_12 <-> RTD Inputs Channel 3/Value

CONFIGURATION Phase0
    RESOURCE PLC ON TwinCAT3
        TASK PlcTask(INTERVAL := T#10ms, PRIORITY := 20);
        PROGRAM MAIN WITH PlcTask : MAIN;
    END_RESOURCE
END_CONFIGURATION

// ---- Data_Types/E_MachineState.TcDUT
// Phase 0 - E_MachineState
// Rev 1.0 - March 13, 2024

TYPE E_MachineState :
(
	eStateOff						:= 0,
	eIdle,
	eHolding,
	eVacant1,
	eRepressurization,
	eAdsorption,
	eEvacuation,
	eDesorption,
	eChangeState,
	eSafeShutdown1,
	eSafeShutdown2,
	eSafeShutdown3,
	ePause
);
END_TYPE

// ---- Data_Types/E_PIDMode.TcDUT
// E_PIDMode
// Rev 1.0 - April 24, 2024

TYPE E_PIDMode :
(
	eOff						:= 0,
	eManual,
	eAuto,
	eTune
);
END_TYPE

// ---- Data_Types/E_Status.TcDUT
// Phase 0 - E_Status
// Rev 1.0 - January 10, 2024

TYPE E_Status :
(
	eSystem_Idle						:= 0,
	e1,
	e2,
	eWarmup_Running,							// 3	
	eSteamBypass_Running,						// 4
	eRepressurization_Running,					// 5
	eAdsorption_Running,						// 6
	eEvacuation_Running,						// 7
	eDesorption_Running,						// 8
	eShutting_Down,								// 9
	ePressureTest_Running,						// 10
	e11,
	e12,
	eWarmup_Error,								// 13
	eSteamBypass_Error,							// 14
	eRepressurization_Error,					// 15
	eAdsorption_Error,							// 16
	eEvacuation_Error,							// 17
	eDesorption_Error,							// 18
	eShutdown_Error,							// 19
	ePressureTest_Error,						// 20
	e21,
	e22,
	eWarmup_Complete,							// 23
	eSteamBypass_Complete,						// 24
	eRepressurization_Complete,					// 25
	eAdsorption_Complete,						// 26
	eEvacuation_Complete,						// 27
	eDesorption_Complete,						// 28
	eShutdown_Complete,							// 29
	ePressureTest_Complete,						// 30
	e31,
	e32,
	eStopping_Process,							// 33
	eResetting,									// 34
	eSaving_Data								// 35
);
END_TYPE

// ---- Data_Types/E_Util_Service_Req.TcDUT
//{attribute 'qualified_only'}
//{attribute 'strict'}
{attribute 'to_string'}

TYPE E_Util_Service_Req :
(
	Off			:= 0,
	On 			:= 1
//	Reset		:= 2
);
END_TYPE

// ---- Data_Types/E_WS_State.TcDUT
// Phase 0 - E_WS_State
// Rev 1.0 - January 8, 2024

TYPE E_WS_State :
(
	eWSIdle			 													:= 0,
	eWSReadCoils,
	eWSReadInputStatus,
	eWSReadRegs,
	eWSReadInputRegs,
	eWSWriteSingleCoil,
	eWSWriteSingleReg,
	eWSWriteMultipleCoils,
	eWSWriteRegs
);
END_TYPE

// ---- Data_Types/E_LMH.TcDUT
// Phase 0 - E_LMH
// Rev 1.0 - March 14, 2024

TYPE E_LMH :
(
	eLow			 													:= 0,
	eMid,
	eHigh
);
END_TYPE

// ---- Data_Types/Module.TcDUT
// Phase 0 - Module
// Rev 1.0 - December 25, 2023

TYPE Module :
STRUCT
	
	condensate_from_cooling_and_purge_lines_lsl					: BOOL;
	condensate_from_cooling_and_purge_lines_lsh					: BOOL;
	                                                	
	condensate_from_cooling_and_purge_lines_pump				: BOOL;
                                                    	
	condensate_flow												: REAL;
	condensate_flow_error										: BOOL;
	steam_manifold_line_pres									: REAL;
	steam_manifold_line_pres_error								: BOOL;
                                                    	
	steam_temp_near_rs1											: REAL;
	steam_temp_near_rs1_error									: BOOL;
	steam_temp_near_rs3											: REAL;
	steam_temp_near_rs3_error									: BOOL;
	condensate_temp												: REAL;
	condensate_temp_error										: BOOL;
	                                                	
END_STRUCT
END_TYPE

// ---- Data_Types/Reactor_Set.TcDUT
// Phase 0 - Reactor_Set
// Rev 1.0 - May 10, 2024

TYPE Reactor_Set :
STRUCT
		
	all_doors_open														: BOOL;
	all_doors_closed													: BOOL;
	all_clamps_extended													: BOOL;
	all_clamps_retracted												: BOOL;
	valves_clear														: BOOL;
	average_reactor_pressure											: REAL;
	average_reactor_pressure_within_ambient								: BOOL;
	reactor_vacuum_status												: INT;
	reactor_pressure_error												: STRING;
    
	condensate_lsl														: BOOL;
	condensate_lsh														: BOOL;
    
	steam_control_valve_position										: REAL;
	steam_control_valve_closed											: BOOL;
	dead_air_valve_clear												: BOOL;
	purge_valve_clear													: BOOL;
	cooling_valve_clear													: BOOL;
	steam_header_valve_clear											: BOOL;
	steam_header_valve_not_closed										: BOOL;
    
	R1_inlet_co2														: REAL;
	R1_outlet_co2														: REAL;
	
	
	
	
	R1_reactor_pres														: REAL;
	R2_reactor_pres														: REAL;
	R3_reactor_pres														: REAL;
	R4_reactor_pres														: REAL;
    
	R1_reactor_pres_error												: BOOL;
	R2_reactor_pres_error												: BOOL;
	R3_reactor_pres_error												: BOOL;
	R4_reactor_pres_error												: BOOL;
	
	repres_valve_error													: STRING;
	
	extend_all_clamps													: BOOL;
	retract_all_clamps													: BOOL;
	open_all_doors														: BOOL;
	close_all_doors														: BOOL;
	close_all_valves													: BOOL;
	co2_sensors_off														: BOOL;
	co2_inside_sensors_on												: BOOL;
	co2_outside_sensors_on												: BOOL;
	open_repres_valves													: BOOL;
	close_repres_valves													: BOOL;
	vacuum_holding														: BOOL;
	
	condensate_pump														: BOOL;
	fan_vfd_percent														: REAL;
	fan_vfd_running														: BOOL;
    
    /// <summary>RS_PCV-01</summary>
	steam_control_valve													: REAL;
	steam_control_valve_mode											: INT;
	steam_control_valve_setpoint										: REAL;
	steam_control_valve_control_point									: REAL;
	dead_air_valve														: BOOL;
    /// <summary>XV-05</summary>
	purge_valve															: BOOL;
    /// <summary>XV-06</summary>
	cooling_valve														: BOOL;
    /// <summary>XV-07</summary>
	steam_header_valve													: BOOL;
    
	desorption_high_temp_count											: INT;
	inlet_air_high_temp_count											: INT;
	vacuum_cooling_high_temp_count										: INT;
	sorbent_high_temp													: REAL;

END_STRUCT
END_TYPE

// ---- Data_Types/ST_Util_Service_Req.TcDUT
TYPE ST_Util_Service_Req :
STRUCT
	rs_number 		: UINT;
	request_cmd		: BOOL;  // (   0 = release/off , 1 = assign/on , 2 =  reset fault)
END_STRUCT
END_TYPE

// ---- Data_Types/ST_Util_Service_Sts.TcDUT
TYPE ST_Util_Service_Sts :
STRUCT  
	idle		: BOOL;
	ready 		: BOOL;
	running		: BOOL;
	faulted		: BOOL;
END_STRUCT
END_TYPE

// ---- Data_Types/Utility.TcDUT
// Phase 0 - STRUCT - Utility
// Rev 1.0 - May 13, 2024

TYPE Utility :
STRUCT

	utility_error														: STRING;
	os_air_unsafe_temp													: BOOL;
	
	safe_shutdown_error_1												: STRING;
	safe_shutdown_error_2												: STRING;
	
	auto_mode_on														: BOOL;
	drainage_on															: BOOL;
	
	product_condensate_drum_lsl											: BOOL;
	product_condensate_drum_lsh											: BOOL;
	condensate_collection_tank_lsl										: BOOL;
	condensate_collection_tank_lsh										: BOOL;
	
	boiler_package														: BOOL;
	boiler_ready														: BOOL;
	product_condensate_pump												: BOOL;
	condensate_collection_tank_pump										: BOOL;
	product_condenser													: BOOL;
	dead_air_vacuum_pump												: BOOL;
	product_blower														: BOOL;
	instrument_air_compressor											: BOOL;
	dead_air_line_co2_pump												: BOOL;
	dead_air_line_co2_sol												: BOOL;
	
	dead_air_line_co2													: REAL;
	dead_air_line_co2_error												: BOOL;
	product_outlet_co2													: REAL;
	product_outlet_co2_error											: BOOL;
	product_outlet_h2o													: REAL;
	product_outlet_h2o_error											: BOOL;
	product_outlet_o2													: REAL;
	product_outlet_o2_error												: BOOL;
	product_co2sample_h2o												: REAL;
	product_co2sample_h2o_error											: BOOL;
	product_outlet_temperature											: REAL;
	product_outlet_temperature_error									: BOOL;
	condensate_collection_tank_ph										: REAL;
	condensate_collection_tank_ph_error									: BOOL;
	condensate_collection_tank_o2										: REAL;
	condensate_collection_tank_o2_error									: BOOL;
	condensate_collection_tank_turbidity								: REAL;
	condensate_collection_tank_turbidity_error							: BOOL;

	dead_air_flow														: REAL;
	dead_air_flow_error													: BOOL;
	product_outlet_volumetric_flow										: REAL;
	product_outlet_volumetric_flow_error								: BOOL;
	product_outlet_mass_flow											: REAL;
	product_outlet_mass_flow_error										: BOOL;
	product_condenser_pump_outlet_liquid_flow							: REAL;
	product_condenser_pump_outlet_liquid_flow_error						: BOOL;
	tap_water_to_boiler_flow											: REAL;
	tap_water_to_boiler_flow_error										: BOOL;
	steam_header_flow													: REAL;
	steam_header_flow_error												: BOOL;
	condensate_collection_tank_flow										: REAL;
	condensate_collection_tank_flow_error								: BOOL;

	weather_humidity													: REAL;
	weather_humidity_error												: BOOL;
	weather_temp														: REAL;
	weather_temp_error													: BOOL;
	weather_pres														: REAL;
	weather_pres_error													: BOOL;
	weather_wind_speed													: REAL;
	weather_wind_speed_error											: BOOL;
	weather_noise_level													: REAL;
	weather_noise_level_error											: BOOL;
	weather_wind_direction												: REAL;
	weather_wind_direction_error										: BOOL;

	product_condensate_drum_level										: REAL;
	product_condensate_drum_level_error									: BOOL;
	condensate_collection_tank_level									: REAL;
	condensate_collection_tank_level_error								: BOOL;

	dead_air_line_pres													: REAL;
	dead_air_line_pres_error											: BOOL;
	purge_product_line_pres												: REAL;
	purge_product_line_pres_error										: BOOL;
	pre_condenser_line_pres												: REAL;
	pre_condenser_line_pres_error										: BOOL;
	post_condenser_line_pres											: REAL;
	post_condenser_line_pres_error										: BOOL;
	product_vacuum_pres													: REAL;
	product_vacuum_pres_error											: BOOL;
	product_outlet_pres													: REAL;
	product_outlet_pres_error											: BOOL;
	boiler_outlet_pres													: REAL;
	boiler_outlet_pres_error											: BOOL;
	instrument_air_comp_pres											: REAL;
	instrument_air_comp_pres_error										: BOOL;
	instrument_air_comp_pres_interlock									: INT;
	
	purge_product_line_temp												: REAL;
	purge_product_line_temp_error										: BOOL;
	pre_condenser_line_temp												: REAL;
	pre_condenser_line_temp_error										: BOOL;
	post_condenser_line_temp											: REAL;
	post_condenser_line_temp_error										: BOOL;
	product_outlet_temp													: REAL;
	product_outlet_temp_error											: BOOL;
	product_condenser_pump_outlet_temp									: REAL;
	product_condenser_pump_outlet_temp_error							: BOOL;
	boiler_outlet_temp													: REAL;
	boiler_outlet_temp_error											: BOOL;
	condensate_collection_tank_temp										: REAL;
	condensate_collection_tank_temp_error								: BOOL;
	condensate_collection_tank_outlet_line_temp							: REAL;
	condensate_collection_tank_outlet_line_temp_error					: BOOL;
	instrument_air_comp_temp											: REAL;
	instrument_air_comp_temp_error										: BOOL;
	instrument_air_comp_temp_interlock									: INT;
	
	/// <summary>XV-01</summary>
	cooling_line_pre_condenser_valve									: BOOL;
    /// <summary>XV-01</summary>
	cooling_line_pre_condenser_valve_clear								: BOOL;

	/// <summary>XV-02</summary>
	purge_product_pre_condenser_valve									: BOOL;
	/// <summary>XV-02</summary>
	purge_product_pre_condenser_valve_clear								: BOOL;

    /// <summary>XV-03</summary>
	product_vacuum_pump_isolation_valve									: BOOL;
    /// <summary>XV-03</summary>
	product_vacuum_pump_isolation_valve_clear							: BOOL;
    /// <summary>XV-03</summary>
	product_vacuum_pump_isolation_valve_closed							: BOOL;
	
	product_vacuum_bypass_valve											: BOOL;
	product_vacuum_bypass_valve_clear									: BOOL;
	
    /// <summary>XV-05</summary>
	product_vacuum_outlet_isolation_valve								: BOOL;
    /// <summary>XV-05</summary>
	product_vacuum_outlet_isolation_valve_clear							: BOOL;

	product_condensate_drain_valve										: BOOL;
	
	steam_bypass_valve													: BOOL;
	steam_bypass_valve_clear											: BOOL;
	
	condensate_collection_tank_pump_outlet_valve						: BOOL;
	condensate_collection_tank_pump_outlet_valve_clear					: BOOL;
	
    /// <summary>PCV-01</summary>
	product_vacuum_backfeed_valve_open									: BOOL;
    /// <summary>PCV-01</summary>
	product_vacuum_backfeed_valve_closed								: BOOL;
    /// <summary>PCV-01</summary>
	product_vacuum_backfeed_valve										: REAL;
    /// <summary>PCV-01</summary>
	product_vacuum_backfeed_valve_setpoint								: REAL;
    /// <summary>PCV-01</summary>
	product_vacuum_backfeed_valve_mode									: INT;								
	
    /// <summary>P-02</summary>
	product_vacuum_pump_vfd												: REAL;
	product_vacuum_pump_vfd_output										: REAL;
	product_vacuum_pump_radiator										: BOOL;
	product_blower_vfd													: REAL;
	product_blower_vfd_output											: REAL;
	
	steam_header_volume_total_enable									: BOOL;
	
	 /// <summary>AT04-Chiller</summary>
	 product_co2_chiller												: BOOL;
	 /// <summary>AT04-Chiller-Pump</summary>
	 product_co2_chiller_pump											: BOOL;
	
END_STRUCT
END_TYPE

// ---- GVLs/Global_Alarms.TcGVL
// Phase 0 - Global_Alarms
// Rev 1.0 - May 14, 2024

VAR_GLOBAL
	
	giAlarmCount														: INT		:= 0;
	gsAlarms															: ARRAY[0.._ALARM_COUNT] OF STRING;
	gsMessages															: ARRAY[0.._ALARM_COUNT] OF STRING;

	gsAmbientPressureError												: STRING	:= 'Ambient pressure error';
	gsAdsorptionAcceptableButNotIdealTimeError							: STRING	:= 'Adsorption time to cool acceptable but not ideal';
	gsAdsorptionTimeOutError											: STRING	:= 'Adsorption - sorbent failed to cool';
	gsAdsorptionUnacceptableTimeError									: STRING	:= 'Adsorption time to cool unacceptable';
	gsAdsorptionInletCo2LowError										: STRING	:= 'Adsorption inlet co2 concentration low';
	gsAirFlowSensorError												: STRING	:= 'Air flow sensor error (FT-01)';
	gsBoilerError														: STRING	:= 'Boiler pressure error';
	gsBoilerOutletPresSensorError										: STRING	:= 'Boiler outlet pressure sensor error (PT-07)';
	gsBoilerOutletTempSensorError										: STRING	:= 'Boiler outlet temperature sensor error (TT-06)';
	gsClampExtendError													: STRING	:= 'Clamp extend error';
	gsClampRetractError													: STRING	:= 'Clamp retract error';
	gsCondensateCollectionDrainError									: STRING	:= 'Condensate collection tank not draining';
	gsCondensateCollectionTankFlowSensorError							: STRING	:= 'Condensate collection tank flow sensor error (FT-07)';
	gsCondensateCollectionTankLevelSensorError							: STRING	:= 'Condensate collection tank level sensor error (LT-02)';
	gsCondensateCollectionTankLshError									: STRING	:= 'Condensate collection tank high limit switch error (LS-06)';
	gsCondensateCollectionTankOutletLineTempSensorError					: STRING	:= 'Condensate collection tank outlet line temperature sensor error (TT-08)';
	gsCondensateCollectionTankO2SensorError								: STRING	:= 'Condensate collection tank o2 sensor error (AT-05)';
	gsCondensateCollectionTankPhSensorError								: STRING	:= 'Condensate collection tank ph sensor error (AT-04)';
	gsCondensateCollectionTankTempSensorError							: STRING	:= 'Condensate collection tank temperature sensor error (TT-07)';
	gsCondensateCollectionTankTurbiditySensorError						: STRING	:= 'Condensate collection tank turbidity sensor error (AT-06)';
	gsCondesateFlowSensorError											: STRING	:= 'Condensate flow sensor error (FT-02)';
	gsCondensateFromCoolingAndPurgeLinesLslError						: STRING	:= 'Condensate from cooling and purge lines low limit switch error (LS-03)';
	gsCondensateLslError												: STRING	:= 'Condensate low limit switch error (LS-01)';
	gsCondensateProductDrainError										: STRING	:= 'Module product/cooling line not draining';	
	gsCondensateTempSensorError											: STRING	:= 'Condensate temperature sensor error (TT-12)';	
	gsCoolingValveError													: STRING	:= 'Cooling valve error (XV-06)';
	gsDeadAirFlowSensorError											: STRING	:= 'Dead air flow sensor error (FT-01)';
	gsDeadAirLineCo2SensorError											: STRING	:= 'Dead air line co2 sensor error (AT-01)';
	gsDeadAirLinePresSensorError										: STRING	:= 'Dead air line pressure sensor error (PT-01)';
	gsDeadAirValveError													: STRING	:= 'Dead air valve error (XV-04)';
	gsDesiredCycleCountError											: STRING	:= 'Desired cycle count error';
	gsDesorptionHighSteamLineTemp										: STRING	:= 'Desorption - High steam line temperature';
	gsDesorptionPurgeLinePressureError									: STRING	:= 'Desorption - Unable to purge';
	gsDoorClampsExtendedError											: STRING	:= 'Door clamps extended';
	gsDoorsNotClosedError												: STRING	:= 'Door not closed error';
	gsDoorsNotOpenError													: STRING	:= 'Door not open error';
	gsFanDiffPresSensorError											: STRING	:= 'Fan differential pressure sensor error (PDT-03)';
	gsFilterDiffPresSensorError											: STRING	:= 'Filter differential pressure sensor error (PDT-01)';
	gsHighTempCountError												: STRING	:= 'High Temp Count Error';
	gsInletAirHighTempCountError										: STRING	:= 'Inlet air high temperature count error';
	gsInletAirTempRangeError											: STRING	:= 'Inlet air temperature range error';
    gsInletCO2SensorError												: STRING	:= 'Inlet CO2 sensor error (AT-01)';
    gsInletH2OSensorError												: STRING	:= 'Inlet H2O sensor error (AT-02)';
	gsInletDoorLeftClampsExtendedError									: STRING	:= 'Left inlet door clamps extended error (XV-01)'; 
	gsInletDoorRightClampsExtendedError									: STRING	:= 'Right inlet door clamps extended error (XV-01)'; 
	gsInstrumentAirCompPresSensorError									: STRING	:= 'Instrument air compressor pressure sensor error (PT-08)';
	gsInstrumentAirCompTempSensorError									: STRING	:= 'Instrument air compressor temperature sensor error (TT-09)';
	gsInsufficientVacuumPressureError									: STRING	:= 'Insufficient vacuum pressure reached';
	gsNoReactorSetsSelected												: STRING	:= 'No reactor sets selected';
    gsOutletCO2SensorError												: STRING	:= 'Outlet CO2 sensor error (AT-03)';
    gsOutletH2OSensorError												: STRING	:= 'Outlet H2O sensor error (AT-04)';
	gsOutletDoorLeftClampsExtendedError									: STRING	:= 'Left outlet door clamps extended error (XV-03)'; 
	gsOutletDoorRightClampsExtendedError								: STRING	:= 'Right outlet door clamps extended error (XV-03)'; 
	gsOutsideTempRangeError												: STRING	:= 'Outside air temperature out of range';
	gsPneumaticLineTempError											: STRING	:= 'Pneumatic line temperature out of range (TT-09)';
	gsPostCondenserLinePresSensorError									: STRING	:= 'Post condenser line pressure sensor error (PT-04)';
	gsPostCondenserLineHighTempError									: STRING	:= 'Post condenser line high temperature error';
	gsPostCondenserLineTempSensorError									: STRING	:= 'Post condenser line temperature sensor error (TT-03)';
	gsPreCondenserLinePresSensorError									: STRING	:= 'Pre condenser line pressure sensor error (PT-03)';
	gsPreCondenserLineTempSensorError									: STRING	:= 'Pre condenser line temperature sensor error (TT-02)';
	gsProductCondensateDrainError										: STRING	:= 'Product condensate not draining';
	gsProductCondensateDrainValveError									: STRING	:= 'Product condensate drain valve error';
	gsProductCondensateDrumLshError										: STRING	:= 'Product condensate drum high limit switch error (LS-02)';
	gsProductCondensateDrumLevelSensorError								: STRING	:= 'Product condensate not draining';
	gsProductCondenserPumpOutletLiquidFlowSensorError					: STRING	:= 'Product condenser pump outlet temperature sensor error (TT-05)';
	gsProductCondenserPumpOutletTempSensorError							: STRING	:= 'Product condenser pump outlet temperature sensor error (TT-05)';
	gsProductOutletH2oSensorError										: STRING	:= 'Product outlet h2o sensor error (AT-07A)';
	gsProductOutletTemperatureSensorError								: STRING	:= 'Product outlet h2o sensor error (AT-07B)';
	gsProductCo2SampleH2oSensorError									: STRING	:= 'Product outlet h2o sensor error (AT-02B)';
	gsProductOutletCo2SensorError										: STRING	:= 'Product outlet co2 sensor error (AT-02A)';
	gsProductOutletO2SensorError										: STRING	:= 'Product outlet o2 sensor error (AT-03)';
	gsProductOutletPresSensorError										: STRING	:= 'Product outlet pressure sensor error (PT-06)';
	gsProductOutletTempSensorError										: STRING	:= 'Product outlet temperature sensor error (TT-04)';
	gsProductOutletMassFlowSensorError									: STRING	:= 'Product outlet mass flow sensor error (FT-03)';
	gsProductOutletVolumetricFlowSensorError							: STRING	:= 'Product outlet volumetric flow sensor error (FT-02)';
	gsProductVacuumBackfeedValveError									: STRING	:= 'Product vacuum backfeed valve error (PCV-01)';
	gsProductVacuumOutletIsoValveError									: STRING	:= 'Product vacuum outlet isolation valve error (XV-05)';
	gsProductVacuumPumpIsoValveError									: STRING	:= 'Product vacuum pump isolation valve error (XV-03)';
	gsProductVacuumPumpError											: STRING	:= 'Product vacuum pump error (P-02) - ';
	gsProductVacuumPresSensorError										: STRING	:= 'Product vacuum pressure sensor error (PT-05)';
	gsPurgeProductLinePresLowError										: STRING	:= 'Purge product line pressure low error';
	gsPurgeProductLinePresSensorError									: STRING	:= 'Purge product line pressure sensor error (PT-02)';
	gsPurgeProductLineTempSensorError									: STRING	:= 'Purge product line temperature sensor error (TT-01)';
	gsPurgeValveError													: STRING	:= 'Purge valve error (XV-05)';
	gsReactorDrainError													: STRING	:= 'Reactor not draining';	
	gsReactorDoorClosingError											: STRING	:= 'Failed to close door valves';									// Complete
	gsReactorDoorOpeningError											: STRING	:= 'Failed to open door valves';									// Complete
	gsReactorsAtAmbientPressure											: STRING	:= 'Reactors at ambient pressure';
	gsReactorPressureAboveAcceptableLevelError							: STRING	:= 'Reactor pressure above acceptable level';
	gsReactorPressureAboveDesiredLevelError								: STRING	:= 'Reactor pressure above desired level';
	gsReactorPresError													: STRING	:= 'Reactor pressure error';
	gsReactorPresSensorError											: STRING	:= 'Reactor pressure sensor error  (PT_01)';
	gsReactorSetFailedToPressurizeError									: STRING	:= 'Reactor set failed to pressurize';
	gsReactorValvesNotClosedError										: STRING	:= 'Reactor valves are not closed';
	gsRepressurizationValveError										: STRING	:= 'Repressurization valve error (XV-02)';	
	gsRepressurizationError												: STRING	:= 'Repressurization error';	
	gsSorbentDiffPresSensorError										: STRING	:= 'Sorbent differential pressure sensor error (PDT-02)';
	gsSorbentTemperatureError											: STRING	:= 'Sorbent temperatures above safe temperature';
	gsSteamBypassMinFlowRateError										: STRING	:= 'Steam bypass minimum flow rate error';
	gsSteamControlValveError											: STRING	:= 'Steam control valve error (PCV-01)';
	gsSteamFailedToPressurizeReactorError								: STRING	:= 'Steam failed to pressurize reactor to purge pressure';
	gsSteamHeaderFlowSensorError										: STRING	:= 'Steam header flow sensor error (FT-06)';
	gsSteamHeaderValveError												: STRING	:= 'Steam header valve error (XV-07)';
	gsSteamManifoldLinePresSensorError									: STRING	:= 'Steam manifold line pressure sensro error (PT_02)';
	gsSteamPressureHighError											: STRING	:= 'High steam pressure';
	gsSteamPressureLowError												: STRING	:= 'Low steam pressure';
	gsSteamTemperatureLowError											: STRING	:= 'Low steam temperature';
	gsSteamTempNearRS01SensorError										: STRING	:= 'Steam temperature near RS01 sensor error (TT-10)';
	gsSteamTempNearRS03SensorError										: STRING	:= 'Steam temperature near RS03 sensor error (TT-11)';
	gsTapWaterToBoilerFlowSensorError									: STRING	:= 'Tap water to boiler flow sensor error';
	gsUnableToEvacuateLinesError										: STRING	:= 'Unable to evacuate lines in time';
	gsVacuumCoolingUnacceptableError									: STRING	:= 'Vacuum cooling temperature reached was unacceptable';
	gsVacuumCoolingAcceptableButNotIdealError							: STRING	:= 'Vacuum cooling temperature reached was acceptable but not ideal';
	gsVacuumPressureUnacceptableError									: STRING	:= 'Vacuum pressure reached was unacceptable';
	gsVacuumPressureAcceptableBotNotIdealError							: STRING	:= 'Vacuum pressure reached was acceptable but not ideal';
	gsWarmupNotRunError													: STRING	:= 'Warmup has not run';
	gsWeatherHumiditySensorError										: STRING	:= 'Weather humidity sensor error (AT-07)';
	gsWeatherPresureSensorError											: STRING	:= 'Weather pressure sensor error (PT-09)';
	gsWeatherWindSpeedSensorError										: STRING	:= 'Weather wind speed sensor error (AT-08)';
	gsWeatherWindDirectionSensorError									: STRING	:= 'Weather wind direction sensor error (WDT-01)';
	gsWeatherTempSensorError											: STRING	:= 'Weather temperature sensor error (TT-10)';
	gsWeatherNoiseLevelSensorError										: STRING	:= 'Weather noise level sensor error (NT-01)';
	gsCoolingLinePreCondeserValveError									: STRING	:= 'Cooling Line Pre Condenser Valve Error U-XV01';
	gsPurgeProductPreCondenserValverError								: STRING	:= 'Purge Product PreCondenser Valve Error U-XV02';
	
	gsMessageTBD			: STRING	:= 'TBD';
	gsAdsorptionCo2LowCheck												: STRING	:= 'Check inlet co2 sensor';
	gsCheckOperation													: STRING	:= 'Check sensor operation';
	gsExtraRepressurizationTimeAllowed									: STRING	:= 'Extra repressurization time allowed';
	gsPressureDropTestCannotRun											: STRING	:= 'Pressure drop test cannot run';
	gsProcessCannotContinue												: STRING	:= 'Process cannot continue';
	gsProcessCannotRun													: STRING	:= 'Process cannot run';
	gsProcessCannotRunAdsorptionWillContinue							: STRING	:= 'Process cannot run - Adsorption will continue';
	gsProcessStopsAtEOA													: STRING	:= 'Process will stop at end of Adsorption';
	gsProcessStopsAtEOC													: STRING	:= 'Process will stop at end of current cycle';
	gsProcessWillContinue												: STRING	:= 'Process will continue';
	gsProcessComplete													: STRING	:= 'Process complete';
	gsProcessRestart													: STRING	:= 'Process will attempt to restart on next cycle';
	gsReactorIsUnderVacuum												: STRING	:= 'Reactor is under vacuum';
	gsReactorSetCannotRun												: STRING	:= 'Reactor set cannot run';
	gsReactorSetWillContinue											: STRING	:= 'Reactor set will continue';
	gsReactorSetWillPause												: STRING	:= 'Reactor set will pause';
	gsReactorSetWillStop												: STRING	:= 'Reactor set will stop';
	gsReactorSetWillStopAtEndOfCycle									: STRING	:= 'Reactor set will stop at end of cycle';
	gsReactorSetsInEvacuationWillContinue								: STRING	:= 'Reactor sets in Evacuation will finish, others will stop';
	gsReactorSetWillStopEvacWillFinishOthersWillCompleteCycle			: STRING	:= 'Reactor set will stop, Evacuation will finish, others will complete cycle';
	gsRunWarmup															: STRING	:= 'Run warm up';													
	gsSafeShutdown1														: STRING	:= 'System will do a Safe Shutdown 1';
	gsSafeShutdown2														: STRING	:= 'System will do a Safe Shutdown 2';
	gsSafeShutdown3														: STRING	:= 'System will do a Safe Shutdown 3';
	gsSorbentDamaged													: STRING	:= 'Sorbent damaged';
	gsSteamBypassWillContinueWOAdsorption								: STRING	:= 'Steam Bypass will continue without Adsorption';
	gsSystemCannotRun													: STRING	:= 'System cannot run';
	gsSystemWillStop													: STRING	:= 'System will stop';
	gsSystemWillStopAfterDesorption										: STRING	:= 'System will stop after Desorption';
	gsUnableToCloseDoors												: STRING	:= 'Unable to close doors';
	gsUnableToEvacuateReactorSet										: STRING	:= 'Unable to evacuate reactor set';
	gsUserProcessRestart												: STRING	:= 'User must restart for process to continue';
	gsWarmupWillContinue												: STRING	:= 'Warm up will continue';													
	gsWarmupWillContinueWOAdsorption									: STRING	:= 'Warm up will continue without Adsorption';

END_VAR

// ---- GVLs/Global_Constants.TcGVL
// Phase 0 - Global_Constants
// Rev 1.0 - June 3, 2024

VAR_GLOBAL CONSTANT
	
	_ALARM_COUNT														: INT		:= 100;
	_DRAIN_TIME															: TIME		:= T#3S;
	_PRODUCT_CONDENSATE_VALVE_TIME										: TIME		:= T#3S;
	_FAN_SPEED_MAX														: REAL		:= 1765;		// Maximum Fan RPM
	_FAN_SPEED_MIN														: REAL		:= 300;			// Minimum Fan RPM
	_PUMP_SPEED_MAX														: REAL		:= 3540;		// Maximum Pump RPM
	_PUMP_SPEED_MIN														: REAL		:= 200;			// Minimum Pump RPM
	_FAN_DELAY_TIME														: INT		:= 2000;
	_FAN_RS_DELAY_TIME													: INT		:= 10000;
	_PROCESS_COMPLETE_TIME												: REAL		:= 2000;
	_PAUSE_TIME															: REAL		:= 2000;
	_VALVE_TIME															: REAL		:= 3000;
	_FAN_SHUTDOWN_TIME													: REAL		:= 10000;
	_VALVE_INCREMENT_TIME												: REAL		:= 250;			// Time period for incremental change in valve position (mSecs)
	_STOPPING_TIME														: REAL		:= 2000;
	_VALVE_CLOSED														: INT		:= 3;
	_VALVE_OPEN															: INT		:= 95;
	
	_CURRENT_208_FACTOR													: REAL		:= 655.34;		// =  32767 counts / 50 amps
	_CURRENT_480_FACTOR													: REAL		:= 218.44;      // = 32767 counts / 150 amps
	_CURRENT_BOILER_FACTOR												: REAL 		:= 40.95 * 2 ;	//  = 32767 / 800 Amps * 2 (double coiled)
	_CURRENT_MODULE_FACTOR												: REAL		:= 81.91;		// 0- 800 amps	
	_PERCENT_FACTOR														: REAL		:= 327.67;		// Factor to convert input to output percentage
	_FAN_RPM_FACTOR														: REAL		:= 17.65;		// Factor to convert fan percent input to rpm output (max rpm / 100)
	_PUMP_RPM_FACTOR													: REAL		:= 35.4;		// Factor to convert pump percent input to rpm output (max rpm / 100)
	_BLOWER_RPM_FACTOR													: REAL      := 34.7;		// product blower rpm = 3470
	_VOLTAGE_208_FACTOR													: REAL		:= 218.44;		// 0- 150 VAC
	_VOLTAGE_480_FACTOR													: REAL		:= 65.53;		// 0 - 500 VAC 
	
	_INLET_AIR_MAX_COUNT												: INT		:= 0;
	_ADSORP_MAX_COUNT													: INT		:= 1;
	_VAC_COOLING_MAX_COUNT												: INT		:= 1;
	_DESORP_MAX_COUNT													: INT		:= 1;
	_HIGH_CART_READINGS_MAX												: INT		:= 2;
	_RETRY_ATTEMPTS														: INT		:= 3;
	_MAX_REACTOR_ERRORS													: INT		:= 3;
	
	_PRESSURE_PERCENT													: REAL		:= 0.9;
	_TEMP_DEADBAND														: REAL		:= 0.5;
	
